// TwinCAT 3 PLC project STELLA1Runtime
// ProgramVersion: 3.1.4023.0
// libraries:
//   Tc2_DataExchange, * (Beckhoff Automation GmbH)
//   Tc2_Math, * (Beckhoff Automation GmbH)
//   Tc2_MC2, * (Beckhoff Automation GmbH)
//   Tc2_MC2_Drive, * (Beckhoff Automation GmbH)
//   Tc2_NC, * (Beckhoff Automation GmbH)
//   Tc2_Standard, * (Beckhoff Automation GmbH)
//   Tc2_System, * (Beckhoff Automation GmbH)
//   Tc2_Utilities, * (Beckhoff Automation GmbH)
//   Tc3_IotBase, * (Beckhoff Automation GmbH)
//   Tc3_Module, * (Beckhoff Automation GmbH)
//   VisuDialogs, * (System)
//   PS_DcUpsEC,2.0,Phoenix Contact GmbH & Co.KG
//   VisuSymbols,3.5.10.0,System
// project tree:
//   DUTs/ E_Blink.TcDUT, E_Horn.TcDUT, E_TCSCommand.TcDUT (not stored), E_TCSErrors.TcDUT (not stored), E_TelescopeMode.TcDUT
//   / GlobalTextList.TcGTLO, PlcTask.TcTTO, Visualization Manager.TcVMO (not stored)
//   GVLs/ GVL_FilterWheel.TcGVL, GVL_Hydraulics.TcGVL (not stored), GVL_Main.TcGVL, GVL_pendant_control.TcGVL, GVL_Safety.TcGVL, GVL_Telescope.TcGVL
//   POUs/ AzimuthElevationControl.TcPOU, CoverControl.TcPOU, DerotatorControl.TcPOU, ElevationControl.TcPOU, FilterWheelControl.TcPOU, FocusControl.TcPOU, HydraulicsControl.TcPOU, MAIN.TcPOU, NasmythControl.TcPOU, PendantControl.TcPOU, SafetyHandling.TcPOU, TelescopeAuxiliary.TcPOU, TelescopeControl.TcPOU, Transformer.TcPOU
//   POUs/FunctionBlocks/ CO_ABERRATION.TcPOU (not stored), CO_REFRACT.TcPOU, FB_ALTAZ2HADEC.TcPOU (not stored), FB_AstroClock.TcPOU (not stored), FB_Axis2.TcPOU, FB_BLINK.TcPOU, FB_ButtonEnable.TcPOU (not stored), FB_Cover.TcPOU, FB_CO_NUTATE.TcPOU, FB_EQ2HOR.TcPOU, FB_EQ2HOR2.TcPOU, FB_EventLog.TcPOU, FB_HADEC2ALTAZ.TcPOU, FB_HOR2EQ.TcPOU, FB_HOR2EQ2.TcPOU (not stored), FB_Horn.TcPOU, FB_InfluxMessage.TcPOU (not stored), FB_LightTimer.TcPOU (not stored), FB_MQTTCommunication.TcPOU, FB_NUTATE.TcPOU (not stored), FB_PRECESS.TcPOU, FB_PRECESS2.TcPOU, FB_PRECESS3.TcPOU, FB_RFTRIG.TcPOU (not stored), FB_SUNPOS.TcPOU (not stored), FB_TimeAverage.TcPOU (not stored), FB_Timer.TcPOU (not stored), FB_TONTP.TcPOU, TelescopeAxisClass.TcPOU
//   POUs/Functions/ ATAN2.TcPOU, CO_REFRACT_FORWARD.TcPOU (not stored), CT2LST.TcPOU (not stored), DateTime2JD.TcPOU, F_Azimuthvelocity.TcPOU, F_DerotatorPosition2.TcPOU, F_Derotatorvelocity.TcPOU, F_Elevationvelocity.TcPOU, F_YREAL.TcPOU, NCError_TO_STRING.TcPOU, PointingModelAzimuth.TcPOU, PointingModelElevation.TcPOU, POLY.TcPOU (not stored), Refraction.TcPOU, TEN.TcPOU
//   VISUs/ Visualization.TcVIS
// real-time tasks:
//   TASK PlcTask: cycle T#10ms, priority 20, ADS port 350
// motion (NC):
//   TASK NC-Task 1 SAF: cycle T#2ms, priority 4, ADS port 501
//   TASK NC-Task 1 SVB: cycle T#10ms, priority 8, ADS port 511
//   AXIS Fokus (id 1)
//     Dynamic: AccelerationMaximum=100, DecelerationMaximum=100, Acceleration=4.5, Deceleration=4.5, Jerk=13.5
//     Velo: RefSearch=0.2, RefSync=0.2, SlowManual=0.1, FastManual=0.5, Maximum=3
//     TargetPosControl: Range=0.1
//     OtherSettings: AllowMotionCmdToSlave=true, PulseDistancePos=1, PulseDistanceNeg=1
//     encoder EncType=4
//       EncPara: ScaleFactorNumerator=0.001, ScaleFactorDenominator=5, MaxCount=#x0000ffff
//         SoftEndMinControl: Enable=true
//         SoftEndMaxControl: Enable=true, Range=100
//         Inc: RefMode=2, RefSoftSyncMask=#x0000ffff
//     drive DrvType=23
//       Analog: VeloReferenz=10.2713178, VeloScale=10, TorqueSetpointScale=10, ScaleFactorActTorque=10
//       TimeComp: TaskDelayCycles=1
//     controller CtrType=1
//       CtrPara: PriorControlFactor=1
//         PosDiffControl: Range=1
//         PID: PosKp=12, CtrlOutputLimit=1
//         Observer: BandWidth=20
//   AXIS Derotator (id 2)
//     General: UnitName=°
//     Dynamic: AccelerationMaximum=20, DecelerationMaximum=20, Acceleration=3.70696, Deceleration=3.70696, Jerk=1.65107
//     Velo: RefSearch=1, RefSync=0.5, SlowManual=0.5, FastManual=5, Fast=11.7222517903646, Maximum=11.7223
//     PositionAreaControl: Range=10
//     TargetPosControl: Range=1, Time=0.1
//     OtherSettings: AllowMotionCmdToSlave=true
//     encoder EncType=8
//       EncPara: ScaleFactorNumerator=0.2, ScaleFactorDenominator=1048576, MaxCount=#xffffffff
//         SoftEndMinControl: Enable=true, Range=-70
//         SoftEndMaxControl: Enable=true, Range=380
//     drive DrvType=9
//       DrvPara: MaxCount=#xffffffff, DriveControlDWord=#x00030100
//         Analog: VeloReferenz=12.894476969401, TorqueSetpointScale=10, ScaleFactorActTorque=0.1
//         TimeComp: TaskDelayCycles=1
//     controller CtrType=1
//       CtrPara: PriorControlFactor=1
//         PosDiffControl: Range=1, Time=0.1
//         Observer: BandWidth=20
//   AXIS Azimuth (id 3)
//     General: UnitName=°
//     Dynamic: AccelerationMaximum=10, DecelerationMaximum=10, Acceleration=3, Deceleration=3, Jerk=1
//     Velo: RefSearch=2, RefSync=1, SlowManual=1, FastManual=5, Fast=798, Maximum=10
//     TargetPosControl: Range=1, Time=0.1
//     OtherSettings: AllowMotionCmdToSlave=true
//     encoder EncType=8
//       EncPara: ScaleFactorNumerator=360, ScaleFactorDenominator=1048576, MaxCount=#xffffffff
//         SoftEndMinControl: Enable=true, Range=-50
//         SoftEndMaxControl: Enable=true, Range=450
//         Inc: RefPosition=180, RefMode=2
//     drive DrvType=9
//       DrvPara: MaxCount=#xffffffff, DriveControlDWord=#x00030100
//         Analog: VeloReferenz=877.8, VeloScale=1.02400649589962, TorqueSetpointScale=10, ScaleFactorActTorque=0.1
//         TimeComp: TaskDelayCycles=1
//     controller CtrType=1
//       CtrPara: PriorControlFactor=1
//         PosDiffControl: Range=3, Time=0.1
//         Observer: BandWidth=20
//   AXIS Elevation (id 4)
//     General: UnitName=°
//     Dynamic: AccelerationMaximum=10, DecelerationMaximum=10, Acceleration=3, Deceleration=3, Jerk=2
//     Velo: RefSearch=0.5, RefSync=0.5, SlowManual=1, FastManual=3, Fast=1026, Maximum=10
//     TargetPosControl: Range=1, Time=0.1
//     OtherSettings: AllowMotionCmdToSlave=true
//     encoder EncType=8
//       EncPara: ScaleFactorNumerator=360, ScaleFactorDenominator=1048576, MaxCount=#xffffffff
//         SoftEndMinControl: Enable=true
//         SoftEndMaxControl: Enable=true, Range=91
//         Inc: RefPosition=73.9885, RefMode=2
//     drive DrvType=9
//       DrvPara: MaxCount=#xffffffff, DriveControlDWord=#x00030100
//         Analog: VeloReferenz=1128.6, VeloScale=1.02400649589962, TorqueSetpointScale=10, ScaleFactorActTorque=0.1
//         TimeComp: TaskDelayCycles=1
//     controller CtrType=1
//       CtrPara: PriorControlFactor=1
//         PosDiffControl: Range=1, Time=0.1
//         Observer: BandWidth=20
//   AXIS FilterWheel (id 5)
//     General: UnitName=°, UnitFlags=#x00000004
//     Dynamic: AccelerationMaximum=1500, DecelerationMaximum=1500, Acceleration=15.2, Deceleration=15.2, Jerk=4.44308
//     Velo: RefSearch=5, RefSync=5, SlowManual=1, FastManual=10, Fast=103.833333333333, Maximum=100
//     TargetPosControl: Range=1
//     OtherSettings: AllowMotionCmdToSlave=true
//     encoder EncType=19
//       EncPara: ScaleFactorNumerator=5, ScaleFactorDenominator=1048576, MaxCount=#xffffffff
//         Inc: RefMode=1, HomingSensorSource=9
//     drive DrvType=16
//       DrvPara: MaxCount=#xffffffff, DriveControlDWord=#x00020000
//         Analog: VeloReferenz=114.216666666667, VeloScale=32, PosScale=5, TorqueSetpointScale=10, ScaleFactorActTorque=0.1
//         TimeComp: TaskDelayCycles=1
//     controller CtrType=1
//       CtrPara: PriorControlFactor=1
//         PosDiffControl: Range=0.2
//         PID: PosKp=3
//         Observer: BandWidth=20
// I/O:
//   DEVICE Gerät 1 (EtherCAT), AmsNetId 5.122.3.233.2.1
//     Klemme 30 (EK1200) [EK1200-5000 EtherCAT Netzteil (2A E-Bus)]
//       Safety Logic (EL6910) [EL6910, TwinSAFE PLC]
//       Safety IN (EL1904) [EL1904, 4 Ch. Safety Input 24V, TwinSAFE]
//         modules: Module 1 (FSOES)
//       Safety OUT (EL2904) [EL2904, 4 Ch. Safety Output 24V, 0.5A, TwinSAFE]
//         modules: Module 1 (FSOES), Module 2 (DO)
//       Power analysis (EL3443) [EL3443 3Ch. Power Measuring]
//       Power0 (EL9410) [EL9410 E-Bus Netzteilklemme (Diagnose)]
//       Main Panel IN (EL1008) [EL1008 8K. Dig. Eingang 24V, 3ms]
//       Hydraulics IN (EL1008) [EL1008 8K. Dig. Eingang 24V, 3ms]
//       Trafo Hydraulics IN (EL1008) [EL1008 8K. Dig. Eingang 24V, 3ms]
//       Main Panel Out (EL2008) [EL2008 8K. Dig. Ausgang 24V, 0.5A]
//       Trafo Hydraulics OUT (EL2008) [EL2008 8K. Dig. Ausgang 24V, 0.5A]
//       Temperature IN (EL3202) [EL3202 2K.Ana. Eingang PT100 (RTD)]
//       Power1 (EL9410) [EL9410 E-Bus Netzteilklemme (Diagnose)]
//       Pendant Control (EL1008) [EL1008 8K. Dig. Eingang 24V, 3ms]
//       Pendant Control2 (EL1008) [EL1008 8K. Dig. Eingang 24V, 3ms]
//       M2 M3 Limit switches (EL1008) [EL1008 8K. Dig. Eingang 24V, 3ms]
//       Cover Limit Switches (EL1008) [EL1008 8K. Dig. Eingang 24V, 3ms]
//       Telescope Hydraulics IN (EL1008) [EL1008 8K. Dig. Eingang 24V, 3ms]
//       Pendant Lights (EL2008) [EL2008 8K. Dig. Ausgang 24V, 0.5A]
//       Lock and Horn (EL2008) [EL2008 8K. Dig. Ausgang 24V, 0.5A]
//       Temperature M2 M1 (EL3064) [EL3064 4K.Ana. Eingang 0-10V]
//       Power2 (EL9410) [EL9410 E-Bus Netzteilklemme (Diagnose)]
//       FocusMotor (EL7342) [EL7342 2K. DC-Motor-Endstufe (50V, 3.5A)]
//       FocusEncoder (EL5101-0010) [EL5101-0010 1K. Inc. Encoder 5V (20 Mio. Inkremente/s)]
//       Cover Motors (EL2008) [EL2008 8K. Dig. Ausgang 24V, 0.5A]
//       Klemme 54 (EK1521) [EK1521 1-Port EtherCAT-Abzweig (FX-MultiMode)]
//         Klemme 55 (EK1501) [EK1501 EtherCAT-Koppler (2A E-Bus, FX-MultiMode, ID-Switch)]
//           FilterWheel (EL7211-0010) [EL7211-0010 1K. MDP742 Servo-Motor-Endstufe mit OCT (50V, 4,5A RMS)]
//           Klemme 57 (EL1008) [EL1008 8K. Dig. Eingang 24V, 3ms]
//           Klemme 58 (EL2008) [EL2008 8K. Dig. Ausgang 24V, 0.5A]
//           ShutterCOM (EL6001) [EL6001 Schnittstelle (RS232)]
//           Klemme 60 (EL3064) [EL3064 4K.Ana. Eingang 0-10V]
//           Klemme 69 (EL3202-0010) [EL3202-0010 2K. Ana. Eingang PT100 (RTD), hochgenau]
//           Klemme 65 (EL9011) [EL9011 Endklemme]
//       Klemme 61 (EK1110) [EK1110 EtherCAT-Verlängerung]
//     Derotator(AX5203-0000-0210) [AX5203-0000-0210 EtherCAT Drive (SoE, 2 Ch.)]
//     Azimuth (AX5125-0000-0214) [AX5125-0000-0214 EtherCAT Drive (SoE, 1 Ch.)]
//     Elevation (AX5125-0000-0214) [AX5125-0000-0214 EtherCAT Drive (SoE, 1 Ch.)]
//     Box 74 (Uninterruptible Power Supply) [QUINT4-UPS/24DC/24DC/40/EC]
// variable links:
//   Device 1 (EtherCAT) <-> Device 1 (EtherCAT)/Term 30 (EK1200)/Safety IN (EL1904)
//     Term 30 (EK1200)/Safety Logic (EL6910)/ConnectionOutputs/TwinSafeGroup1.Safety IN (EL1904) - Module 1 (FSOES)_10 RxPDO <-> Module 1 (FSOES)/TxPDO/FSOE
//   Device 1 (EtherCAT) <-> Device 1 (EtherCAT)/Term 30 (EK1200)/Safety Logic (EL6910)
//     Term 30 (EK1200)/Safety IN (EL1904)/Module 1 (FSOES)/RxPDO/FSOE <-> ConnectionInputs/TwinSafeGroup1.Safety IN (EL1904) - Module 1 (FSOES)_10 TxPDO
//     Term 30 (EK1200)/Safety OUT (EL2904)/Module 1 (FSOES)/TxPDO/FSOE <-> ConnectionOutputs/TwinSafeGroup1.Safety OUT (EL2904) - Module 1 (FSOES)_11 RxPDO
//   Device 1 (EtherCAT) <-> Device 1 (EtherCAT)/Term 30 (EK1200)/Safety OUT (EL2904)
//     Term 30 (EK1200)/Safety Logic (EL6910)/ConnectionInputs/TwinSafeGroup1.Safety OUT (EL2904) - Module 1 (FSOES)_11 TxPDO <-> Module 1 (FSOES)/RxPDO/FSOE
//   NC-Task 1 SAF/Axes/Azimuth <-> Device 1 (EtherCAT)/Azimuth (AX5125-0000-0214)
//     Drive/Inputs/In/nDataIn1 <-> AT/Following distance
//     Drive/Inputs/In/nDcOutputTime <-> InfoData/DcOutputShift
//     Drive/Inputs/In/nState1 <-> AT/Drive status word @bit 8
//     Drive/Inputs/In/nState2 <-> AT/Drive status word
//     Drive/Inputs/In/nState4 @bit 1 <-> WcState/InputToggle
//     Drive/Inputs/In/nState4 <-> WcState/WcState
//     Drive/Outputs/Out/nCtrl1 <-> MDT/Master control word @bit 8
//     Drive/Outputs/Out/nDataOut1 <-> MDT/Position command value
//     Enc/Inputs/In/nDataIn1 <-> AT/Position feedback 1 value
//     Enc/Inputs/In/nDataIn3 <-> AT/Probe value 1 positive edge
//     Enc/Inputs/In/nDcInputTime <-> InfoData/DcInputShift
//     Enc/Inputs/In/nState4 @bit 1 <-> WcState/InputToggle
//     Enc/Inputs/In/nState4 <-> WcState/WcState
//     Enc/Inputs/In/nState5 <-> AT/Probe 1 positive latched
//     Enc/Outputs/Out/nCtrl5 <-> MDT/Probe 1 enable
//   NC-Task 1 SAF/Axes/Derotator <-> Device 1 (EtherCAT)/Derotator(AX5203-0000-0210)
//     Drive/Inputs/In/nDataIn1 <-> AT 1/Following distance
//     Drive/Inputs/In/nDataIn3[0] <-> AT 1/Torque/force feedback value
//     Drive/Inputs/In/nDcOutputTime <-> InfoData/DcOutputShift
//     Drive/Inputs/In/nState1 <-> AT 1/Drive status word @bit 8
//     Drive/Inputs/In/nState2 <-> AT 1/Drive status word
//     Drive/Inputs/In/nState4 @bit 1 <-> WcState/InputToggle
//     Drive/Inputs/In/nState4 <-> WcState/WcState
//     Drive/Outputs/Out/nCtrl1 <-> MDT 1/Master control word @bit 8
//     Drive/Outputs/Out/nDataOut1 <-> MDT 1/Position command value
//     Enc/Inputs/In/nDataIn1 <-> AT 1/Position feedback 1 value
//     Enc/Inputs/In/nDcInputTime <-> InfoData/DcInputShift
//     Enc/Inputs/In/nState4 @bit 1 <-> WcState/InputToggle
//     Enc/Inputs/In/nState4 <-> WcState/WcState
//   NC-Task 1 SAF/Axes/Elevation <-> Device 1 (EtherCAT)/Elevation (AX5125-0000-0214)
//     Drive/Inputs/In/nDataIn1 <-> AT/Following distance
//     Drive/Inputs/In/nDcOutputTime <-> InfoData/DcOutputShift
//     Drive/Inputs/In/nState1 <-> AT/Drive status word @bit 8
//     Drive/Inputs/In/nState2 <-> AT/Drive status word
//     Drive/Inputs/In/nState4 @bit 1 <-> WcState/InputToggle
//     Drive/Inputs/In/nState4 <-> WcState/WcState
//     Drive/Outputs/Out/nCtrl1 <-> MDT/Master control word @bit 8
//     Drive/Outputs/Out/nDataOut1 <-> MDT/Position command value
//     Enc/Inputs/In/nDataIn1 <-> AT/Position feedback 1 value
//     Enc/Inputs/In/nDataIn3 <-> AT/Probe value 1 positive edge
//     Enc/Inputs/In/nDcInputTime <-> InfoData/DcInputShift
//     Enc/Inputs/In/nState4 @bit 1 <-> WcState/InputToggle
//     Enc/Inputs/In/nState4 <-> WcState/WcState
//     Enc/Inputs/In/nState5 <-> AT/Probe 1 positive latched
//     Enc/Outputs/Out/nCtrl5 <-> MDT/Probe 1 enable
//   NC-Task 1 SAF/Axes/FilterWheel <-> Device 1 (EtherCAT)/Term 30 (EK1200)/Term 54 (EK1521)/Term 55 (EK1501)/FilterWheel (EL7211-0010)
//     Drive/Inputs/In/nDcOutputTime <-> InfoData/DcOutputShift
//     Drive/Inputs/In/nState1 <-> DRV Statusword/Statusword
//     Drive/Inputs/In/nState2 <-> DRV Statusword/Statusword @bit 8
//     Drive/Inputs/In/nState4 @bit 1 <-> WcState/InputToggle
//     Drive/Inputs/In/nState4 <-> WcState/WcState
//     Drive/Inputs/In/nState8 <-> DRV Info data 1/Info data 1
//     Drive/Outputs/Out/nCtrl1 <-> DRV Controlword/Controlword
//     Drive/Outputs/Out/nCtrl2 <-> DRV Controlword/Controlword @bit 8
//     Drive/Outputs/Out/nDataOut2 <-> DRV Target velocity/Target velocity
//     Enc/Inputs/In/nDataIn1 <-> FB Position/Position
//     Enc/Inputs/In/nDcInputTime <-> InfoData/DcInputShift
//     Enc/Inputs/In/nState4 @bit 1 <-> WcState/InputToggle
//     Enc/Inputs/In/nState4 <-> WcState/WcState
//   NC-Task 1 SAF/Axes/Fokus <-> Device 1 (EtherCAT)/Term 30 (EK1200)/FocusEncoder (EL5101-0010)
//     Enc/Inputs/In/nDataIn1[0] <-> ENC Status compact/Counter value
//     Enc/Inputs/In/nDataIn2[0] <-> ENC Status compact/Latch value
//     Enc/Inputs/In/nState1 <-> ENC Status compact/Status/Latch C valid
//     Enc/Inputs/In/nState1 @bit 1 <-> ENC Status compact/Status/Latch extern valid
//     Enc/Inputs/In/nState1 @bit 6 <-> ENC Status compact/Status/Open circuit
//     Enc/Inputs/In/nState1 @bit 2 <-> ENC Status compact/Status/Set counter done
//     Enc/Inputs/In/nState1 @bit 5 <-> ENC Status compact/Status/Status of input status
//     Enc/Inputs/In/nState2 @bit 4 <-> ENC Status compact/Status/Status of extern latch
//     Enc/Inputs/In/nState2 <-> ENC Status compact/Status/Status of input A
//     Enc/Inputs/In/nState2 @bit 1 <-> ENC Status compact/Status/Status of input B
//     Enc/Inputs/In/nState2 @bit 2 <-> ENC Status compact/Status/Status of input C
//     Enc/Inputs/In/nState2 @bit 3 <-> ENC Status compact/Status/Status of input gate
//     Enc/Inputs/In/nState2 @bit 5 <-> ENC Status compact/Status/Sync error
//     Enc/Inputs/In/nState2 @bit 6 <-> ENC Status compact/Status/TxPDO State
//     Enc/Inputs/In/nState2 @bit 7 <-> ENC Status compact/Status/TxPDO Toggle
//     Enc/Inputs/In/nState4 @bit 1 <-> WcState/InputToggle
//     Enc/Inputs/In/nState4 <-> WcState/WcState
//     Enc/Outputs/Out/nCtrl1 <-> ENC Control compact/Control/Enable latch C
//     Enc/Outputs/Out/nCtrl1 @bit 3 <-> ENC Control compact/Control/Enable latch extern on negative edge
//     Enc/Outputs/Out/nCtrl1 @bit 1 <-> ENC Control compact/Control/Enable latch extern on positive edge
//     Enc/Outputs/Out/nCtrl1 @bit 2 <-> ENC Control compact/Control/Set counter
//     Enc/Outputs/Out/nDataOut1[0] <-> ENC Control compact/Set counter value
//   NC-Task 1 SAF/Axes/Fokus <-> Device 1 (EtherCAT)/Term 30 (EK1200)/FocusMotor (EL7342)
//     Drive/Inputs/In/nState1 @bit 3 <-> DCM Status Channel 1/Status/Error
//     Drive/Inputs/In/nState1 @bit 5 <-> DCM Status Channel 1/Status/Moving negative
//     Drive/Inputs/In/nState1 @bit 4 <-> DCM Status Channel 1/Status/Moving positive
//     Drive/Inputs/In/nState1 @bit 1 <-> DCM Status Channel 1/Status/Ready
//     Drive/Inputs/In/nState1 <-> DCM Status Channel 1/Status/Ready to enable
//     Drive/Inputs/In/nState1 @bit 6 <-> DCM Status Channel 1/Status/Torque reduced
//     Drive/Inputs/In/nState1 @bit 2 <-> DCM Status Channel 1/Status/Warning
//     Drive/Inputs/In/nState2 @bit 3 <-> DCM Status Channel 1/Status/Digital input 1
//     Drive/Inputs/In/nState2 @bit 4 <-> DCM Status Channel 1/Status/Digital input 2
//     Drive/Inputs/In/nState2 @bit 5 <-> DCM Status Channel 1/Status/Sync error
//     Drive/Inputs/In/nState2 @bit 7 <-> DCM Status Channel 1/Status/TxPDO Toggle
//     Drive/Inputs/In/nState4 @bit 1 <-> WcState/InputToggle
//     Drive/Inputs/In/nState4 <-> WcState/WcState
//     Drive/Outputs/Out/nCtrl1 <-> DCM Control Channel 1/Control/Enable
//     Drive/Outputs/Out/nCtrl1 @bit 2 <-> DCM Control Channel 1/Control/Reduce torque
//     Drive/Outputs/Out/nCtrl1 @bit 1 <-> DCM Control Channel 1/Control/Reset
//     Drive/Outputs/Out/nCtrl1 @bit 3 <-> DCM Control Channel 1/Control/Threshold active
//     Drive/Outputs/Out/nDataOut2[0] <-> DCM Velocity Channel 1/Velocity
//   STELLA1Runtime/STELLA1Runtime Instance <-> Device 1 (EtherCAT)/Azimuth (AX5125-0000-0214)
//     PlcTask Inputs/GVL_Telescope.Azimuth_diagnostic <-> AT/Diagnostic number
//     PlcTask Inputs/GVL_Telescope.Azimuth_inputs <-> AT/Digital inputs, state
//     PlcTask Inputs/GVL_Telescope.Azimuth_torque <-> AT/Torque/force feedback value
//   STELLA1Runtime/STELLA1Runtime Instance <-> Device 1 (EtherCAT)/Box 74 (Uninterruptible Power Supply)
//     PlcTask Inputs/MAIN.arrInputPD @bit {304..432 step 32} <-> TxPDO 1/BATTERY {1..5} ALARMS  (5 links)
//     PlcTask Inputs/MAIN.arrInputPD @bit 80 <-> TxPDO 1/STATUS ACTUAL INPUT CURRENT
//     PlcTask Inputs/MAIN.arrInputPD @bit 64 <-> TxPDO 1/STATUS ACTUAL INPUT VOLTAGE
//     PlcTask Inputs/MAIN.arrInputPD @bit 112 <-> TxPDO 1/STATUS ACTUAL OUTPUT CURRENT 1
//     PlcTask Inputs/MAIN.arrInputPD @bit 96 <-> TxPDO 1/STATUS ACTUAL OUTPUT VOLTAGE 1
//     PlcTask Inputs/MAIN.arrInputPD @bit 128 <-> TxPDO 1/STATUS BATTERY ACTUAL VOLTAGE
//     PlcTask Inputs/MAIN.arrInputPD @bit 144 <-> TxPDO 1/STATUS BATTERY CHARGE CURRENT
//     PlcTask Inputs/MAIN.arrInputPD @bit 160 <-> TxPDO 1/STATUS BATTERY TEMPERATURE
//     PlcTask Inputs/MAIN.arrInputPD @bit 176 <-> TxPDO 1/STATUS DEVICE TEMPERATURE
//     PlcTask Inputs/MAIN.arrInputPD <-> TxPDO 1/STATUS FUNCTIONS
//     PlcTask Inputs/MAIN.arrInputPD @bit 32 <-> TxPDO 1/STATUS INTERFACE
//     PlcTask Inputs/MAIN.arrInputPD @bit 192 <-> TxPDO 1/STATUS SOC REMAINING TIME
//     PlcTask Inputs/MAIN.arrInputPD @bit 224 <-> TxPDO 1/STATUS SOC REMAINING TIME PC SHUTDOWN
//     PlcTask Inputs/MAIN.arrInputPD @bit 240 <-> TxPDO 1/STATUS SOH REMAINING LIFETIME
//     PlcTask Inputs/MAIN.arrInputPD @bit 272 <-> TxPDO 1/UPS DIAGNOSIS ALARMS
//     PlcTask Inputs/MAIN.arrInputPD @bit 256 <-> TxPDO 1/UPS PROCESS ALARMS
//   STELLA1Runtime/STELLA1Runtime Instance <-> Device 1 (EtherCAT)/Derotator(AX5203-0000-0210)
//     PlcTask Inputs/GVL_Telescope.Derotator_diagnostic <-> AT 1/Diagnostic number
//     PlcTask Inputs/GVL_Telescope.Derotator_inputs <-> AT 1/Digital inputs, state
//     PlcTask Inputs/GVL_Telescope.Derotator_torque <-> AT 1/Torque/force feedback value
//   STELLA1Runtime/STELLA1Runtime Instance <-> Device 1 (EtherCAT)/Elevation (AX5125-0000-0214)
//     PlcTask Inputs/GVL_Telescope.Elevation_diagnostic <-> AT/Diagnostic number
//     PlcTask Inputs/GVL_Telescope.Elevation_inputs <-> AT/Digital inputs, state
//     PlcTask Inputs/GVL_Telescope.Elevation_torque <-> AT/Torque/force feedback value
//   STELLA1Runtime/STELLA1Runtime Instance <-> Device 1 (EtherCAT)/Term 30 (EK1200)/Cover Limit Switches (EL1008)
//     PlcTask Inputs/GVL_Telescope.cover1_closed <-> Channel 2/GVL_Telescope.cover1_closed
//     PlcTask Inputs/GVL_Telescope.cover2_closed <-> Channel 4/GVL_Telescope.cover2_closed
//     PlcTask Inputs/GVL_Telescope.cover3_closed <-> Channel 6/GVL_Telescope.cover3_closed
//     PlcTask Inputs/GVL_Telescope.cover1_open <-> Channel 1/GVL_Telescope.cover1_open
//     PlcTask Inputs/GVL_Telescope.cover2_open <-> Channel 3/GVL_Telescope.cover2_open
//     PlcTask Inputs/GVL_Telescope.cover3_open <-> Channel 5/GVL_Telescope.cover3_open
//   STELLA1Runtime/STELLA1Runtime Instance <-> Device 1 (EtherCAT)/Term 30 (EK1200)/Cover Motors (EL2008)
//     PlcTask Outputs/GVL_Telescope.close_cover1 <-> Channel 4/GVL_Telescope.close_cover1
//     PlcTask Outputs/GVL_Telescope.close_cover2 <-> Channel 6/GVL_Telescope.close_cover2
//     PlcTask Outputs/GVL_Telescope.close_cover3 <-> Channel 8/GVL_Telescope.close_cover3
//     PlcTask Outputs/GVL_Telescope.nasmyth_left <-> Channel 1/GVL_Telescope.nasmyth_left
//     PlcTask Outputs/GVL_Telescope.nasmyth_right <-> Channel 2/GVL_Telescope.nasmyth_right
//     PlcTask Outputs/GVL_Telescope.open_cover1 <-> Channel 3/GVL_Telescope.open_cover1
//     PlcTask Outputs/GVL_Telescope.open_cover2 <-> Channel 5/GVL_Telescope.open_cover2
//     PlcTask Outputs/GVL_Telescope.open_cover3 <-> Channel 7/GVL_Telescope.open_cover3
//   STELLA1Runtime/STELLA1Runtime Instance <-> Device 1 (EtherCAT)/Term 30 (EK1200)/Hydraulics IN (EL1008)
//     PlcTask Inputs/GVL_Hydraulics.oil_high <-> Channel 2/GVL_Hydraulics.oil_high
//     PlcTask Inputs/GVL_Hydraulics.oil_low <-> Channel 1/GVL_Hydraulics.oil_low
//     PlcTask Inputs/GVL_Hydraulics.oil_overtemperature <-> Channel 4/GVL_Hydraulics.oil_overtemperature
//     PlcTask Inputs/GVL_Hydraulics.oil_pressure_OK <-> Channel 3/GVL_Hydraulics.oil_pressure_OK
//     PlcTask Inputs/GVL_Hydraulics.oil_undertemperature <-> Channel 5/GVL_Hydraulics.oil_undertemperature
//     PlcTask Inputs/GVL_Hydraulics.oilfilter_dirty <-> Channel 6/GVL_Hydraulics.oilfilter_dirty
//   STELLA1Runtime/STELLA1Runtime Instance <-> Device 1 (EtherCAT)/Term 30 (EK1200)/Lock and Horn (EL2008)
//     PlcTask Outputs/GVL_Telescope.focus_unlock <-> Channel 1/GVL_Telescope.focus_lock
//     PlcTask Outputs/GVL_Telescope.horn <-> Channel 8/GVL_Telescope.horn
//     PlcTask Outputs/GVL_Telescope.nasmyth_lock <-> Channel 2/GVL_Telescope.nasmyth_lock
//   STELLA1Runtime/STELLA1Runtime Instance <-> Device 1 (EtherCAT)/Term 30 (EK1200)/M2 M3 Limit switches (EL1008)
//     PlcTask Inputs/GVL_Telescope.focus_limit_far <-> Channel 2/GVL_Telescope.focus_limit_far
//     PlcTask Inputs/GVL_Telescope.focus_limit_near <-> Channel 1/GVL_Telescope.focus_limit_near
//     PlcTask Inputs/GVL_Telescope.nasmyth_limit_left <-> Channel 3/GVL_Telescope.nasmyth_limit_left
//     PlcTask Inputs/GVL_Telescope.nasmyth_limit_right <-> Channel 4/GVL_Telescope.nasmyth_limit_right
//   STELLA1Runtime/STELLA1Runtime Instance <-> Device 1 (EtherCAT)/Term 30 (EK1200)/Main Panel IN (EL1008)
//     PlcTask Inputs/GVL_Main.key_switch_remote <-> Channel 1/GVL_Main.key_switch_remote
//     PlcTask Inputs/GVL_Main.reset_switch <-> Channel 4/GVL_Main.reset_switch
//     PlcTask Inputs/GVL_Main.start_switch <-> Channel 2/GVL_Main.start_switch
//     PlcTask Inputs/GVL_Main.stop_switch <-> Channel 3/GVL_Main.stop_switch
//   STELLA1Runtime/STELLA1Runtime Instance <-> Device 1 (EtherCAT)/Term 30 (EK1200)/Main Panel Out (EL2008)
//     PlcTask Outputs/GVL_Main.lamp_error <-> Channel 3/GVL_Main.lamp_error
//     PlcTask Outputs/GVL_Main.lamp_on_manual <-> Channel 2/GVL_Main.lamp_ready
//     PlcTask Outputs/GVL_Main.lamp_power <-> Channel 1/GVL_Main.lamp_power
//   STELLA1Runtime/STELLA1Runtime Instance <-> Device 1 (EtherCAT)/Term 30 (EK1200)/Pendant Control (EL1008)
//     PlcTask Inputs/GVL_pendant_control.BCD1 <-> Channel 1/GVL_pendant_control.BCD1
//     PlcTask Inputs/GVL_pendant_control.BCD2 <-> Channel 2/GVL_pendant_control.BCD2
//     PlcTask Inputs/GVL_pendant_control.BCD4 <-> Channel 3/GVL_pendant_control.BCD4
//     PlcTask Inputs/GVL_pendant_control.BCD8 <-> Channel 4/GVL_pendant_control.BCD8
//     PlcTask Inputs/GVL_pendant_control.direction_down <-> Channel 7/GVL_pendant_control.direction_down
//     PlcTask Inputs/GVL_pendant_control.direction_up <-> Channel 6/GVL_pendant_control.direction_up
//     PlcTask Inputs/GVL_pendant_control.key_switch <-> Channel 8/GVL_pendant_control.key_switch
//     PlcTask Inputs/GVL_pendant_control.reset_switch <-> Channel 5/GVL_pendant_control.reset_switch
//   STELLA1Runtime/STELLA1Runtime Instance <-> Device 1 (EtherCAT)/Term 30 (EK1200)/Pendant Control2 (EL1008)
//     PlcTask Inputs/GVL_pendant_control.direction_left <-> Channel 2/GVL_pendant_control.direction_left
//     PlcTask Inputs/GVL_pendant_control.direction_right <-> Channel 3/GVL_pendant_control.direction_right
//     PlcTask Inputs/GVL_pendant_control.start_switch <-> Channel 1/GVL_pendant_control.start_switch
//   STELLA1Runtime/STELLA1Runtime Instance <-> Device 1 (EtherCAT)/Term 30 (EK1200)/Pendant Lights (EL2008)
//     PlcTask Outputs/GVL_pendant_control.lamp_down <-> Channel 2/GVL_pendant_control.lamp_down
//     PlcTask Outputs/GVL_pendant_control.lamp_error <-> Channel 5/GVL_pendant_control.lamp_error
//     PlcTask Outputs/GVL_pendant_control.lamp_left <-> Channel 4/GVL_pendant_control.lamp_left
//     PlcTask Outputs/GVL_pendant_control.lamp_right <-> Channel 3/GVL_pendant_control.lamp_right
//     PlcTask Outputs/GVL_pendant_control.lamp_up <-> Channel 1/GVL_pendant_control.lamp_up
//   STELLA1Runtime/STELLA1Runtime Instance <-> Device 1 (EtherCAT)/Term 30 (EK1200)/Safety Logic (EL6910)
//     PlcTask Inputs/GVL_Safety.Error <-> StandardInputs/TwinSafeGroup1.SafetyError_4
//     PlcTask Inputs/GVL_Safety.State <-> Function Block Info Data/TwinSafeGroup1.Network1.FBEstop1 Info Data/State
//     PlcTask Inputs/GVL_Safety.Stop <-> StandardInputs/TwinSafeGroup1.SafetyStop_7
//     PlcTask Outputs/GVL_Safety.ErrAck <-> StandardOutputs/TwinSafeGroup1.ErrorAcknowledgement_1
//     PlcTask Outputs/GVL_Safety.Restart <-> StandardOutputs/TwinSafeGroup1.RestartSafety_2
//     PlcTask Outputs/GVL_Safety.Run <-> StandardOutputs/TwinSafeGroup1.RunSafety_3
//   STELLA1Runtime/STELLA1Runtime Instance <-> Device 1 (EtherCAT)/Term 30 (EK1200)/Telescope Hydraulics IN (EL1008)
//     PlcTask Inputs/GVL_Hydraulics.oil_reserve <-> Channel 2/GVL_Hydraulics.oil_reserve
//     PlcTask Inputs/GVL_Hydraulics.oilpan_maximum <-> Channel 1/GVL_Hydraulics.oilpan_maximum
//     PlcTask Inputs/GVL_Telescope.azimut_limit_switch <-> Channel 8/GVL_Telescope.azimut_limit_switch
//   STELLA1Runtime/STELLA1Runtime Instance <-> Device 1 (EtherCAT)/Term 30 (EK1200)/Temperature IN (EL3202)
//     PlcTask Inputs/GVL_Main.main_cabinet_temperature <-> RTD Inputs Channel 1/Value
//   STELLA1Runtime/STELLA1Runtime Instance <-> Device 1 (EtherCAT)/Term 30 (EK1200)/Temperature M2 M1 (EL3064)
//     PlcTask Inputs/GVL_Telescope.temperature_mirror1 <-> AI Standard Channel 2/Value
//     PlcTask Inputs/GVL_Telescope.temperature_mirror2 <-> AI Standard Channel 1/Value
//   STELLA1Runtime/STELLA1Runtime Instance <-> Device 1 (EtherCAT)/Term 30 (EK1200)/Term 54 (EK1521)/Term 55 (EK1501)/FilterWheel (EL7211-0010)
//     PlcTask Inputs/GVL_FilterWheel.bCalibrationCam <-> DRV Info data 1/Info data 1
//   STELLA1Runtime/STELLA1Runtime Instance <-> Device 1 (EtherCAT)/Term 30 (EK1200)/Term 54 (EK1521)/Term 55 (EK1501)/Term 60 (EL3064)
//     PlcTask Inputs/TelescopeAuxiliary.raw_dewar_pressure <-> AI Standard Channel 1/Value
//   STELLA1Runtime/STELLA1Runtime Instance <-> Device 1 (EtherCAT)/Term 30 (EK1200)/Trafo Hydraulics IN (EL1008)
//     PlcTask Inputs/GVL_Hydraulics.pump_running <-> Channel 7/GVL_Hydraulics.pump_running
//     PlcTask Inputs/GVL_Hydraulics.suction_running <-> Channel 8/GVL_Hydraulics.suction_running
//     PlcTask Inputs/GVL_Main.brake_clearing <-> Channel 3/GVL_Main.brake_clearing
//     PlcTask Inputs/GVL_Main.trafo_bypassed <-> Channel 2/GVL_Main.trafo_bypassed
//   STELLA1Runtime/STELLA1Runtime Instance <-> Device 1 (EtherCAT)/Term 30 (EK1200)/Trafo Hydraulics OUT (EL2008)
//     PlcTask Outputs/GVL_Hydraulics.oil_pump_enable <-> Channel 1/GVL_Hydraulics.oil_pump_enable
//     PlcTask Outputs/GVL_Hydraulics.oil_suction_enable <-> Channel 2/GVL_Hydraulics.oil_suction_enable
//     PlcTask Outputs/GVL_Main.softstart_trafo <-> Channel 8/GVL_Main.softstart_trafo
//     PlcTask Outputs/GVL_Telescope.brake_azimuth_eve <-> Channel 3/GVL_Telescope.brake_azimuth_eve
//   STELLA1Runtime/STELLA1Runtime Instance <-> NC-Task 1 SAF/Axes/Azimuth
//     PlcTask Inputs/GVL_Telescope.AzimuthAxisRef.NcToPlc <-> Outputs/ToPlc
//     PlcTask Outputs/GVL_Telescope.AzimuthAxisRef.PlcToNc <-> Inputs/FromPlc
//   STELLA1Runtime/STELLA1Runtime Instance <-> NC-Task 1 SAF/Axes/Derotator
//     PlcTask Inputs/GVL_Telescope.DerotatorAxisRef.NcToPlc <-> Outputs/ToPlc
//     PlcTask Outputs/GVL_Telescope.DerotatorAxisRef.PlcToNc <-> Inputs/FromPlc
//   STELLA1Runtime/STELLA1Runtime Instance <-> NC-Task 1 SAF/Axes/Elevation
//     PlcTask Inputs/GVL_Telescope.ElevationAxisRef.NcToPlc <-> Outputs/ToPlc
//     PlcTask Outputs/GVL_Telescope.ElevationAxisRef.PlcToNc <-> Inputs/FromPlc
//   STELLA1Runtime/STELLA1Runtime Instance <-> NC-Task 1 SAF/Axes/FilterWheel
//     PlcTask Inputs/GVL_FilterWheel.FilterWheel_AxisRef.NcToPlc <-> Outputs/ToPlc
//     PlcTask Outputs/GVL_FilterWheel.FilterWheel_AxisRef.PlcToNc <-> Inputs/FromPlc
//   STELLA1Runtime/STELLA1Runtime Instance <-> NC-Task 1 SAF/Axes/Fokus
//     PlcTask Inputs/GVL_Telescope.FocusAxisRef.NcToPlc <-> Outputs/ToPlc
//     PlcTask Outputs/GVL_Telescope.FocusAxisRef.PlcToNc <-> Inputs/FromPlc

CONFIGURATION STELLA1Runtime
    RESOURCE PLC ON TwinCAT3
        TASK PlcTask(INTERVAL := T#10ms, PRIORITY := 20);
        PROGRAM MAIN WITH PlcTask : MAIN;
    END_RESOURCE
END_CONFIGURATION

// ---- DUTs/E_Blink.TcDUT
{attribute 'qualified_only'}
{attribute 'strict'}
TYPE E_Blink :
(
	off := 0,
	slow,
	fast,
	short,
	long,
	on
);
END_TYPE

// ---- DUTs/E_Horn.TcDUT
{attribute 'qualified_only'}
{attribute 'strict'}
TYPE E_Horn :
(
	off := 0,
	beep,
	short,
	long
);
END_TYPE

// ---- DUTs/E_TelescopeMode.TcDUT
{attribute 'qualified_only'}
{attribute 'strict'}
TYPE E_TelescopeMode :
(
	off := 0,
	manual := 1,
	automatic := 2
);
END_TYPE

// ---- GVLs/GVL_FilterWheel.TcGVL
{attribute 'qualified_only'}
VAR_GLOBAL
	FilterWheel_AxisRef:	AXIS_REF;
	bCalibrationCam			AT%I*:	BOOL;
END_VAR

// ---- GVLs/GVL_Main.TcGVL
{attribute 'qualified_only'}
//TODO update to current RoboTel IOs
VAR_GLOBAL
	//DIN1 0.0
	//phase_available		AT%I*: BOOL;
	// not implemented on stella
	trafo_bypassed		AT%I*: BOOL;
	//not implemented on RoboTel
	//key_switch			AT%I*: BOOL;
	//DIN3 0.2
	key_switch_remote	AT%I*: BOOL;
	//DIN4 0.3
	start_switch		AT%I*: BOOL;
	//DIN5 0.4
	stop_switch			AT%I*: BOOL;
	//DIN8 0.7
	reset_switch		AT%I*: BOOL;
	
	//BT1
	main_cabinet_temperature	AT%I*: INT;
	//DIN15 1.6
	brake_clearing		AT%I*: BOOL;
	
	//DOUT1 0.0
	lamp_power			AT%Q*: BOOL;
	//DOUT2 0.1
	lamp_on_manual			AT%Q*: BOOL;
	//DOUT3 0.2
	lamp_error			AT%Q*: BOOL;
	
	//DOUT7 0.6
	softstart_trafo		AT%Q*:BOOL;

	isRoboTel:		BOOL;
END_VAR

// ---- GVLs/GVL_pendant_control.TcGVL
{attribute 'qualified_only'}
//TODO update to current RoboTel IOs
VAR_GLOBAL
	//DIN17 2.0
	BCD1		AT%I*: BOOL;
	//DIN18 2.1
	BCD2		AT%I*: BOOL;
	//DIN19 2.2
	BCD4		AT%I*: BOOL;
	//DIN20 2.3
	BCD8		AT%I*: BOOL;
	//DIN21 2.4
	reset_switch	AT%I*: BOOL;
	//DIN22 2.5
	direction_up	AT%I*: BOOL;
	//DIN23 2.6
	direction_down	AT%I*: BOOL;
	//DIN24 2.7
	key_switch		AT%I*: BOOL;
	//DIN25 3.0 (enable)
	start_switch	AT%I*: BOOL;
	//DIN26 3.1
	direction_left	AT%I*: BOOL;
	//DIN27 3.2
	direction_right	AT%I*: BOOL;
	
	// Outputs
	
	//DOUT9 1.0
	lamp_up			AT%Q*: BOOL;
	//DOUT10 1.1
	lamp_down			AT%Q*: BOOL;
	//DOUT11 1.2
	lamp_right			AT%Q*: BOOL;
	//DOUT12 1.3
	lamp_left			AT%Q*: BOOL;
	//DOUT13 1.4
	lamp_error			AT%Q*: BOOL;
	
END_VAR

// ---- GVLs/GVL_Safety.TcGVL
{attribute 'qualified_only'}
VAR_GLOBAL
	// Safety Error Condition
	Error		AT%I*:	BOOL;
	// Run/Stop Safety
	Run			AT%Q*:	BOOL;
	// Restart Safety
	Restart		AT%Q*:	BOOL;
	// Error Acknowledgement 
	ErrAck		AT%Q*:	BOOL;
	// Stop signal coming from Safety
	Stop		AT%I*:	BOOL;
END_VAR

// ---- GVLs/GVL_Telescope.TcGVL
{attribute 'qualified_only'}
VAR_GLOBAL
	// BT9 mirror
	temperature_mirror2		AT%I*: INT;
	// BT10
	temperature_mirror1		AT%I*: INT;

	//DOUT6 0.5
	brake_azimuth_eve	AT%Q*: BOOL;
	
	// DIN28 3.3 (absolute)
	azimut_limit_switch	AT%I*: BOOL;
	// DIN29 3.4
	focus_limit_near	AT%I*: BOOL;
	// DIN30 3.5
	focus_limit_far		AT%I*: BOOL;
	// DIN31 3.6
	nasmyth_limit_left	AT%I*: BOOL;
	// DIN32 3.7
	nasmyth_limit_right	AT%I*: BOOL;
	
	// DIN33 4.0
	cover1_open		AT%I*: BOOL;
	// DIN34 4.1
	cover1_closed	AT%I*: BOOL;
	// DIN35 4.2
	cover2_open		AT%I*: BOOL;
	// DIN36 4.3
	cover2_closed	AT%I*: BOOL;
	// DIN37 4.4
	cover3_open		AT%I*: BOOL;
	// DIN38 4.5
	cover3_closed	AT%I*: BOOL;

	//DOUT14 1.5
	focus_unlock		AT%Q*: BOOL;
	//DOUT15 4.6
	nasmyth_lock	AT%Q*: BOOL;
	//Horn 4.7
	horn			AT%Q*: BOOL;
	
	// digitale inputs der Endlagen
	Derotator_inputs		AT%I*: WORD;
	// diagnostic number
	Derotator_diagnostic	AT%I*: UDINT;
	// derotator torque feedback
	Derotator_torque		AT%I*: INT;
	
	// digital inputs for limit switches
	Elevation_inputs		AT%I*: WORD;
	// diagnostic number
	Elevation_diagnostic	AT%I*: UDINT;
	// torque feedback
	Elevation_torque		AT%I*: INT;
	
	// digital inputs for limit switches
	Azimuth_inputs			AT%I*: WORD;
	// diagnostic number
	Azimuth_diagnostic		AT%I*: UDINT;
	// torque feedback
	Azimuth_torque			AT%I*: INT;
	
	// Zyklisches Interface zwischen NC und Achse
	AzimuthAxisRef: 	AXIS_REF;
	ElevationAxisRef: 	AXIS_REF;
	DerotatorAxisRef: 	AXIS_REF;
 	// Motor1 Channel 1
	FocusAxisRef:		AXIS_REF;
	
	nasmyth_left	AT%Q*: BOOL;
	nasmyth_right	AT%Q*: BOOL;
	open_cover1		AT%Q*: BOOL;
	close_cover1	AT%Q*: BOOL;
	open_cover2		AT%Q*: BOOL;
	close_cover2	AT%Q*: BOOL;
	open_cover3		AT%Q*: BOOL;
	close_cover3	AT%Q*: BOOL;
	
	
END_VAR

// ---- POUs/MAIN.TcPOU
PROGRAM MAIN
VAR
	// telescope drives are ready to enable
	ready:				BOOL;
	// error stat on drive, power or hydraulics
	error:				BOOL;
	// manual, panel or remote reset
	reset:				BOOL;
	// start hydraulics
	start:				BOOL;
	// stop hydraulics 
	stop:				BOOL;
	// soft start trafo
	key_switch:			BOOL;
	//	open brake
	brake_clearing:		BOOL := FALSE;
	
	remote_start:		BOOL;
	remote_stop: 		BOOL;
	remote_reset:		BOOL;
	remote_keyswitch:	BOOL;
	remote_brake_clearing:	BOOL;
	// blink error lamp on warning
	error_lamp: 		FB_BLINK;
	power_lamp:			FB_BLINK;
	sound_horn:			FB_Horn;
	// main cabinet temperature in degrees
	cabinet_temperature:	REAL;
	// measures time between soft start command and power available
	ups_output_voltage:		REAL;
	ups_output_current:		REAL;
	ups_output_power:		REAL;
	PhaseLog:				FB_EventLog;
	TemperatureEvent,
	TemperatureCriticalEvent:	FB_EventLog;
	MQTTTimer : 		TON := (PT:=T#5S);
	GetHostName:		FB_GetHostName;
	HostName: 			STRING(255);
//	LightSwitch:		FB_ButtonEnable;
//	Lightbutton: 		BOOL;
	bExecute:			BOOL := TRUE;
	cabinet_temperature_warning:	SR;
	cabinet_temperature_critical:	SR;
	MQTTClient:		FB_MQTTCommunication;
	ups: 				PS_Q4_DcUpsEC_Cyclic_2;
	xActivate:			BOOL := TRUE;
	arrInputPD	AT%I*:	ARRAY[0..30] OF WORD;
	UPS_Error,
	UPS_Alarm,
	UPS_Warning,
	UPS_BatMode,
	UPS_ReplaceBattery:	FB_EventLog;
END_VAR

(* 
Main control loop
* Execute sub modules
* power management
* control panel switches and status lamps

* start switch activates Hydraulics and Trafo
* 
*)
GetHostName(bExecute := bExecute, sHostName => HostName);
bExecute := FALSE;
start := GVL_Main.start_switch OR remote_start;
stop := (NOT GVL_Main.stop_switch) OR remote_stop;
key_switch := GVL_Main.key_switch_remote OR remote_keyswitch;
brake_clearing := GVL_Main.brake_clearing OR remote_brake_clearing;
reset := GVL_Main.reset_switch OR GVL_pendant_control.reset_switch OR remote_reset;		
brake_clearing := NOT GVL_Main.brake_clearing;
cabinet_temperature := INT_TO_REAL(GVL_Main.main_cabinet_temperature) / 10.0;
cabinet_temperature_warning(SET1 := cabinet_temperature > 50.0,
							RESET := cabinet_temperature < 40.0);
cabinet_temperature_critical(SET1 := cabinet_temperature > 60.0,
							RESET := cabinet_temperature < 50.0);
IF key_switch THEN
	Transformer.start();
ELSE
	Transformer.stop();
END_IF

IF reset THEN
	Transformer.reset();
END_IF

IF start THEN
	HydraulicsControl.enable := TRUE;
END_IF
IF stop THEN
	HydraulicsControl.enable := FALSE;
END_IF

// telescope is ready when power available
ready :=  GVL_main.trafo_bypassed;

// QUINT UPS control section
ups(
	xActivate:= xActivate, 
	arrInputPD:= arrInputPD, 
	xActive=> , 
	xError=> , 
	wDiagCode=> , 
	wAddDiagCode=> , 
	wOutputVoltage=> ups_output_voltage, 
	wOutputCurrent=> ups_output_current, 
	xBatModeActive=> , 
	udtDataStruct=> , 
	xAlarm=> , 
	xWarning=> , 
	xReplaceBattery=> , 
	udtDiag=> );
	
ups_output_voltage := ups_output_voltage / 1000.0;
ups_output_current := ups_output_current / 1000.0;
ups_output_power := ups_output_voltage * ups_output_current;
		
TelescopeControl();	//
CoverControl();	//
PendantControl();	//
NasmythControl();	//
HydraulicsControl();	//
ElevationControl();	//
AzimuthElevationControl();	//
DerotatorControl();	//
FilterWheelControl();	//
FocusControl();
MQTTClient();
Transformer();

error := GVL_Telescope.azimut_limit_switch
			OR FilterWheelControl.Error
			OR Focuscontrol.Error
			OR NasmythControl.error
			OR CoverControl.Error;
// set control lights					
GVL_Main.lamp_on_manual := PendantControl.manual;

IF GVL_Safety.Error THEN
	error_lamp.blink := e_blink.short;
ELSIF ElevationControl.error OR AzimuthElevationControl.error OR DerotatorControl.Error THEN
	error_lamp.blink := e_blink.long;
ELSIF HydraulicsControl.oil_warning OR HydraulicsControl.oil_hot OR HydraulicsControl.pressure_failure THEN
	error_lamp.blink := e_blink.slow;
ELSIF Transformer.error THEN
	error_lamp.blink := e_blink.fast;
ELSIF error THEN
	error_lamp.blink := e_blink.on;
ELSE
	error_lamp.blink := e_blink.off; 
END_IF

IF Transformer.restart_inhibited THEN
	power_lamp.blink := e_blink.short;
ELSIF GVL_main.trafo_bypassed THEN 
	power_lamp.blink := e_blink.on;
ELSIF Transformer.phase_available THEN
	power_lamp.blink := e_blink.long;
ELSIF NOT Transformer.phase_available THEN
	power_lamp.blink := e_blink.off;
ELSIF  Transformer.error THEN
	power_lamp.blink := e_blink.fast;
ELSE 
	power_lamp.blink := e_blink.off; 
END_IF
error_lamp(Q => GVL_Main.lamp_error);
//GVL_Main.lamp_error := error_lamp.Q;
power_lamp(Q => GVL_Main.lamp_power);
//GVL_Main.lamp_power := power_lamp.Q;

IF GVL_Telescope.azimut_limit_switch THEN
	sound_horn.horn := E_horn.long;
ELSIF Hydraulicscontrol.suction_failure THEN
	sound_horn.horn := E_horn.long;
ELSIF TelescopeControl.poweronwarning.Q THEN
	sound_horn.horn := E_horn.short;
ELSIF Pendantcontrol.horn THEN
	sound_horn.horn := E_horn.beep;
ELSE
	sound_horn.horn := E_horn.off;
END_IF 

sound_horn(Q => GVL_Telescope.horn );

SafetyHandling();

MQTTTimer(IN:=TRUE);
IF MQTTTimer.Q THEN // publish new payload every second
	MQTTTimer(IN:=FALSE);
	MQTTClient.Publish('electronics', 'base', 'MainCabinetTemperature', LREAL_TO_FMTSTR(cabinet_temperature, 2, TRUE));
	MQTTClient.Publish('electronics', 'base', 'PowerOK', BOOL_TO_STRING(Transformer.power_ok));
	MQTTClient.Publish('electronics', 'base', 'PhaseOK', BOOL_TO_STRING(Transformer.phase_available));
	MQTTClient.Publish('electronics', 'base', 'MainReady', BOOL_TO_STRING(ready));
	MQTTClient.Publish('electronics', 'base', 'MasterError', BOOL_TO_STRING(error));
	MQTTClient.Publish('electronics', 'base', 'UPSOutputVoltage', LREAL_TO_FMTSTR(ups_output_voltage, 3, TRUE));
	MQTTClient.Publish('electronics', 'base', 'UPSOutputCurrent', LREAL_TO_FMTSTR(ups_output_current, 3, TRUE));
	MQTTClient.Publish('electronics', 'base', 'UPSOutputPower', LREAL_TO_FMTSTR(ups_output_power, 3, TRUE));
	MQTTClient.Publish('electronics', 'base', 'UpsError', BOOL_TO_STRING(ups.xError));
	MQTTClient.Publish('electronics', 'base', 'UpsAlarm', BOOL_TO_STRING(ups.xAlarm));
	MQTTClient.Publish('electronics', 'base', 'UpsWarning', BOOL_TO_STRING(ups.xWarning));
	MQTTClient.Publish('electronics', 'base', 'UpsBatteryMode', BOOL_TO_STRING(ups.xBatModeActive));
	MQTTClient.Publish('electronics', 'base', 'UPSReplaceBattery', BOOL_TO_STRING(ups.xReplaceBattery));
END_IF

PhaseLog(	
	Trigger := 		NOT Transformer.phase_available, 
	Level := 		ADSLOG_MSGTYPE_ERROR,
	FormatString :=	'%s',
	OnMessage := 	'electrical phases:	ERROR!',
	OffLevel := 	ADSLOG_MSGTYPE_HINT,
	OffMEssage := 	'electrical phases:	active');
	
TemperatureEvent(	
	Trigger := 		cabinet_temperature_warning.Q1, 
	Level := 		ADSLOG_MSGTYPE_WARN,
	FormatString :=	'Main cabinet temperature warning:	%s',
	OnMessage := 	LREAL_TO_FMTSTR( cabinet_temperature, 1, TRUE),);
TemperatureCriticalEvent(	
	Trigger := 		cabinet_temperature_critical.Q1, 
	Level := 		ADSLOG_MSGTYPE_ERROR,
	FormatString :=	'Main cabinet temperature is critical:	%s!',
	OnMessage := 	LREAL_TO_FMTSTR( cabinet_temperature, 1, TRUE),);
	
UPS_Error(	
	Trigger := 		ups.xError, 
	Level := 		ADSLOG_MSGTYPE_ERROR,
	OnMessage := 	'UPS has an error!');

UPS_Alarm(	
	Trigger := 		ups.xAlarm, 
	Level := 		ADSLOG_MSGTYPE_ERROR,
	OnMessage := 	'UPS has an alarm!');

	
UPS_Warning(	
	Trigger := 		ups.xWarning, 
	Level := 		ADSLOG_MSGTYPE_WARN,
	OnMessage := 	'UPS has a warning!');

UPS_BatMode(	
	Trigger := 		ups.xBatModeActive, 
	Level := 		ADSLOG_MSGTYPE_WARN,
	OnMessage := 	'UPS is on battery!');

UPS_ReplaceBattery(	
	Trigger := 		ups.xReplaceBattery, 
	Level := 		ADSLOG_MSGTYPE_WARN,
	OnMessage := 	'Replace UPS battery!');

END_PROGRAM

// ---- POUs/FunctionBlocks/FB_BLINK.TcPOU
FUNCTION_BLOCK FB_BLINK
VAR_INPUT
	blink:		E_Blink;
	ON_TIME:	TIME := T#500MS;
	OFF_TIME:	TIME := T#500MS;
END_VAR
VAR_OUTPUT
	Q:		BOOL;
END_VAR
VAR
    IMPULS   :TOF;
    PAUSE    :TOF;
END_VAR

CASE blink OF
	e_blink.off:
		ON_TIME := T#0MS;
		OFF_TIME := T#1000MS;
	e_blink.slow:
		ON_TIME := T#500MS;
		OFF_TIME := T#500MS;
	e_blink.fast:
		ON_TIME := T#250MS;
		OFF_TIME := T#250MS;
	e_blink.short:
		ON_TIME := T#100MS;
		OFF_TIME := T#900MS;
	e_blink.long:
		ON_TIME := T#900MS;
		OFF_TIME := T#100MS;
	e_blink.on:
		ON_TIME := T#0MS;
		OFF_TIME := T#0MS;
END_CASE

IMPULS(IN:= NOT PAUSE.Q AND NOT IMPULS.Q, PT:= ON_TIME);
PAUSE(IN:= NOT PAUSE.Q AND NOT IMPULS.Q, PT:= OFF_TIME);
IF blink = e_blink.off THEN
	Q := FALSE;
ELSIF blink = e_blink.on THEN
	Q := TRUE;
ELSE
	Q := IMPULS.Q;	
END_IF

END_FUNCTION_BLOCK

// ---- POUs/FunctionBlocks/FB_Horn.TcPOU
FUNCTION_BLOCK FB_Horn
VAR_INPUT
	horn:	E_Horn;
END_VAR
VAR_OUTPUT
		Q:		BOOL;
END_VAR
VAR
	ON_TIME:	TIME := T#500MS;
	IMPULS   :TOF;
    PAUSE    :TOF;

END_VAR

CASE horn OF
	e_horn.off:
		ON_TIME := T#0MS;
	e_horn.beep:
		ON_TIME := T#500MS;
	e_horn.short:
		ON_TIME := T#3000MS;
	e_horn.long:
		ON_TIME := T#5000MS;
END_CASE

IMPULS(IN:= NOT PAUSE.Q AND NOT IMPULS.Q, PT:= ON_TIME);
IF horn = e_horn.off THEN
	Q := FALSE;
ELSE
	Q := IMPULS.Q;	
END_IF

END_FUNCTION_BLOCK

// ---- POUs/FunctionBlocks/FB_EventLog.TcPOU
FUNCTION_BLOCK FB_EventLog
VAR_INPUT
	Trigger:		BOOL;
	// ADSLOG_MSGTYPE_HINT or ADSLOG_MSGTYPE_WARN or ADSLOG_MSGTYPE_ERROR
	Level:			UDINT := ADSLOG_MSGTYPE_HINT;
	FormatString: 	STRING(255) := '%s';
	OnMessage: 		STRING(255) := '';
	OffMessage:		STRING(255) := '';
	OffLevel:		UDINT := ADSLOG_MSGTYPE_HINT;
END_VAR
VAR_OUTPUT
END_VAR
VAR
	LogonTrigger: R_TRIG;
	LogoffTrigger: F_TRIG; // R_Trig or F_Trig ?!
	sPayloadPub, PayloadMessage: STRING(255);
	fbFormat:	FB_FormatString;
END_VAR

LogonTrigger(CLK := Trigger);
LogoffTrigger(CLK := Trigger);
// in case the OffLevel is not set use the default Level Value
IF OffLevel = 0 THEN
	OffLevel := Level;
END_IF
IF LogonTrigger.Q AND LEN(OnMessage)>0 THEN
	ADSLOGSTR( Level OR ADSLOG_MSGTYPE_LOG, FormatString, OnMessage);
END_IF

IF LogoffTrigger.Q AND LEN(OffMessage)>0 THEN
	ADSLOGSTR( OffLevel OR ADSLOG_MSGTYPE_LOG, FormatString, OffMessage);
END_IF

sPayloadPub := 'log,host=CX-22747A';

IF LogonTrigger.Q AND LEN(OnMessage)>1 THEN
	IF Level=ADSLOG_MSGTYPE_HINT THEN
		sPayloadPub := CONCAT(sPayloadPub, ',level=INFO');
	ELSIF Level=ADSLOG_MSGTYPE_WARN THEN
		sPayloadPub := CONCAT(sPayloadPub, ',level=WARNING');
	ELSE
	    sPayloadPub := CONCAT(sPayloadPub, ',level=ERROR');
	END_IF
	fbFormat( sFormat := FormatString, arg1 := F_STRING(OnMessage), sOut => PayloadMessage);
	sPayloadPub := APPEND(sPayloadPub, ' message="', PayloadMessage);
	sPayloadPub := CONCAT(sPayloadPub, '"');
	MQTTCommunication.fbMqttClient.Publish(	
					sTopic:= 'STELLA1/Log', 
					pPayload:= ADR(sPayloadPub), 
					nPayloadSize:= LEN2(ADR(sPayloadPub)),
					eQoS:= TcIotMqttQos.AtMostOnceDelivery,
					bRetain:= FALSE, 
					bQueue:= FALSE );
END_IF

IF LogoffTrigger.Q AND LEN(OffMessage)>1 THEN
	IF OffLevel=ADSLOG_MSGTYPE_HINT THEN
		sPayloadPub := CONCAT(sPayloadPub, ',level=INFO');
	ELSIF OffLevel=ADSLOG_MSGTYPE_WARN THEN
		sPayloadPub := CONCAT(sPayloadPub, ',level=WARNING');
	ELSE
	    sPayloadPub := CONCAT(sPayloadPub, ',level=ERROR');
	END_IF
	
	fbFormat( sFormat := FormatString, arg1 := F_STRING(OffMessage), sOut => PayloadMessage);
	sPayloadPub := APPEND(sPayloadPub, ' message="', PayloadMessage);
	sPayloadPub := CONCAT(sPayloadPub, '"');
	MQTTCommunication.fbMqttClient.Publish(	
					sTopic:= 'STELLA1/Log', 
					pPayload:= ADR(sPayloadPub), 
					nPayloadSize:= LEN2(ADR(sPayloadPub)),
					eQoS:= TcIotMqttQos.AtMostOnceDelivery,
					bRetain:= FALSE, 
					bQueue:= FALSE );
END_IF

END_FUNCTION_BLOCK

// ---- POUs/FunctionBlocks/FB_MQTTCommunication.TcPOU
FUNCTION_BLOCK FB_MQTTCommunication
VAR_INPUT
END_VAR
VAR_OUTPUT
END_VAR
VAR
	GetHostName:		FB_GetHostName;
	HostName: 			STRING(255);
    bSetParameter:		BOOL := FALSE;
    bConnect:			BOOL := FALSE;
    (* received message *)
	bSubscribed: 		BOOL;
	sTopicSub: 			STRING(255) := 'STELLA1/Telescope/SET';
	{attribute 'TcEncoding':='UTF-8'}
	sTopicRcv: 			STRING(255);
	{attribute 'TcEncoding':='UTF-8'}
	fbMessageQueue:		FB_IotMqttMessageQueue;
    fbMessage:			FB_IotMqttMessage;
	fbMqttClient:		FB_IotMqttClient;
	sPayloadRcv: 		STRING;
	influxMessage:		FB_InfluxMessage;
	measurement, 
	parameter, 
	value:		STRING(255);
END_VAR

(*
MQTT Communication section

Source:
https://infosys.beckhoff.com/english.php?content=../content/1033/tf6701_tc3_iot_communication_mqtt/3518541195.html&id=

*)
IF HostName='' THEN
	GetHostName.bExecute := TRUE;
ELSE
	GetHostName.bExecute := FALSE;
	bSetParameter := TRUE;
END_IF

GetHostName(sHostName => HostName);

// set the parameters once
IF bSetParameter THEN
    bSetParameter               := FALSE;
    fbMqttClient.sHostName      := 'sky.stella.iac.es';
    fbMqttClient.nHostPort      := 1883;
    fbMqttClient.sClientId      := HostName; 
    fbMqttClient.sTopicPrefix   := ''; 
	fbMqttClient.nKeepAlive     := 60; 
    fbMqttClient.ipMessageQueue := fbMessageQueue;
	bConnect := TRUE;
END_IF

// connect to the client
IF NOT fbMqttClient.bConnected THEN
;
END_IF

fbMqttClient.Execute(bConnect);
	
IF fbMqttClient.bConnected THEN
    IF NOT bSubscribed THEN
        bSubscribed := fbMqttClient.Subscribe(sTopic:=sTopicSub, 
												eQoS:=TcIotMqttQos.AtMostOnceDelivery);
    END_IF
END_IF

// receive queued messages
IF fbMessageQueue.nQueuedMessages > 0 THEN
    IF fbMessageQueue.Dequeue(fbMessage:=fbMessage) THEN
        fbMessage.GetTopic(pTopic:=ADR(sTopicRcv), nTopicSize:=SIZEOF(sTopicRcv) );
        fbMessage.GetPayload(pPayload:=ADR(sPayloadRcv), nPayloadSize:=SIZEOF(sPayloadRcv), bSetNullTermination:=TRUE);
		ADSLOGSTR( ADSLOG_MSGTYPE_HINT OR ADSLOG_MSGTYPE_LOG, 'MQTT %s', sPayloadRcv);
		IF sTopicRcv = sTopicSub THEN
			influxMessage(  sPayload := sPayloadRcv, measurement => measurement, parameter => parameter, value => value);
			IF NOT PendantControl.manual AND measurement = 'command' THEN
				IF parameter = 'power' THEN
					TelescopeControl.power := STRING_TO_BOOL(value);
				ELSIF parameter = 'park' THEN
					TelescopeControl.park := STRING_TO_BOOL(value);
				ELSIF parameter = 'gohome' THEN
					TelescopeControl.gohome := STRING_TO_BOOL(value);
				ELSIF parameter = 'track' THEN
					TelescopeControl.track := STRING_TO_BOOL(value);
				ELSIF parameter = 'goto' THEN
					TelescopeControl.goto := STRING_TO_BOOL(value);
				ELSIF parameter = 'slew' THEN
					TelescopeControl.slew := STRING_TO_BOOL(value);
				ELSIF parameter = 'stop' THEN
					TelescopeControl.stop := STRING_TO_BOOL(value);
				ELSIF parameter = 'reset' THEN
					TelescopeControl.reset := STRING_TO_BOOL(value);
				ELSIF parameter = 'masterreset' THEN
					ElevationControl.bSoEReset := STRING_TO_BOOL(value);
					AzimuthElevationControl.bSoEReset := STRING_TO_BOOL(value);
					DerotatorControl.bSoEReset := STRING_TO_BOOL(value);
				ELSIF parameter = 'nasmyth' THEN
					NasmythControl.left := STRING_TO_USINT(value) = 1;
					NasmythControl.right := STRING_TO_USINT(value) = 2;
				ELSIF parameter = 'rightascension' THEN
					TelescopeControl.track := FALSE;
					TelescopeControl.rightascension := STRING_TO_LREAL(value);
				ELSIF parameter = 'declination' THEN
					TelescopeControl.track := FALSE;
					TelescopeControl.declination := STRING_TO_LREAL(value);
				ELSIF parameter = 'elevation' THEN
					TelescopeControl.elevation := STRING_TO_LREAL(value);
				ELSIF parameter = 'azimuth' THEN
					TelescopeControl.azimuth := STRING_TO_LREAL(value);
				ELSIF parameter = 'focus' THEN
					FocusControl.position := STRING_TO_LREAL(value);
				ELSIF parameter = 'filter' THEN
					FilterWheelControl.filter_position := STRING_TO_USINT(value);
				ELSIF parameter = 'derotator' THEN
					TelescopeControl.track := FALSE;
					TelescopeControl.derotator_offset := STRING_TO_LREAL(value);
				ELSIF parameter = 'elevationoffset' THEN
					TelescopeControl.elevation_offset := STRING_TO_LREAL(value);
				ELSIF parameter = 'azimuthoffset' THEN
					TelescopeControl.azimuth_offset := STRING_TO_LREAL(value);
				ELSIF parameter = 'derotatoroffset' THEN
					TelescopeControl.derotator_offset := STRING_TO_LREAL(value);ELSE
					ADSLOGSTR( ADSLOG_MSGTYPE_WARN OR ADSLOG_MSGTYPE_LOG, 'MQTT not understood %s', sPayloadRcv);
				END_IF
			END_IF // measurement
		END_IF // Topic
		sPayloadRcv := '';
    END_IF // Dequeue
END_IF

PROPERTY Error : BOOL
GET
Error := fbMqttClient.bError;
END_GET
END_PROPERTY

METHOD Publish : BOOL
VAR_INPUT
	domain: 	STRING(255) := 'environment';
	location: 	STRING(255) := 'roof';
	parameter:	STRING(255);
	value:		STRING(255);
END_VAR
VAR
	sPayloadPub: STRING(255) := '';
	fbFormat:	FB_FormatString;
	bError:		BOOL;
	nErrID: UDINT;
	retain_message:		BOOL := FALSE;
END_VAR
//sPayloadPub := 'environment,location=roof,host=CX-4E6032 ';
fbFormat( sFormat := '%s,location=%s,host=%s %s=%s', 
			arg1 := F_STRING(domain), 
			arg2 := F_STRING(location), 
			arg3 := F_STRING(HostName),
			arg4 := F_STRING(parameter),
			arg5 := F_STRING(value),
 
			sOut => sPayloadPub,
			bError => bError, 
			nErrID => nErrID );
// retain message if value is boolean
retain_message := value = 'TRUE' OR value = 'FALSE';

Publish := fbMqttClient.Publish(	
				sTopic:= 'STELLA1/Telemetry', 
				pPayload:= ADR(sPayloadPub), 
				nPayloadSize:= LEN2(ADR(sPayloadPub)),
				eQoS:= TcIotMqttQos.AtMostOnceDelivery,
				bRetain:= retain_message, 
				bQueue:= FALSE );
END_METHOD

METHOD PublishLog : BOOL
VAR_INPUT
	level: 	STRING(255) := 'INFO';
	message:	STRING(255);
	
END_VAR
VAR
	sPayloadPub: STRING(255) := '';
	fbFormat:	FB_FormatString;
	bError:		BOOL;
	nErrID: UDINT;
END_VAR
VAR_OUTPUT
	published: BOOL;
END_VAR
//sPayloadPub := 'environment,location=roof,host=CX-4E6032 ';
fbFormat( sFormat := 'log,host=%s,level=%s message="%s"', 
			arg1 := F_STRING(HostName), 
			arg2 := F_STRING(level), 
			arg3 := F_STRING(message),
 
			sOut => sPayloadPub,
			bError => bError, 
			nErrID => nErrID );

published := fbMqttClient.Publish(	
				sTopic:= 'STELLA1/Log', 
				pPayload:= ADR(sPayloadPub), 
				nPayloadSize:= LEN2(ADR(sPayloadPub)),
				eQoS:= TcIotMqttQos.AtMostOnceDelivery,
				bRetain:= FALSE, 
				bQueue:= FALSE );
END_METHOD

END_FUNCTION_BLOCK

// ---- POUs/PendantControl.TcPOU
PROGRAM PendantControl
VAR
	// program selection of the pendant control
	Selection:	UINT;
	// error on the pendant control
	Error:		BOOL;
	// manual switch
	manual:		BOOL;
	//enable button
	enable:		BOOL;
	//reset button
	reset:		BOOL;
	// up button
	up:			BOOL;
	// down button
	down:		BOOL;
	// left button
	left:		BOOL;
	// right button
	right:		BOOL;
	lamp_left:		BOOL;
	lamp_right:		BOOL;
	lamp_up:		BOOL;
	lamp_down:		BOOL;
	lamp_error:		BOOL;
	horn:			BOOL;
	// counter for filter position
	Filter_position:	USINT;
	FocusEnable: 		FB_ButtonEnable;
	DerotatorEnable:	FB_ButtonEnable;
	ElevationEnable: 	FB_ButtonEnable;
	AzimuthEnable: 		FB_ButtonEnable;
	FilterWheelEnable:	FB_ButtonEnable;
	TelescopeControlEnable: 	FB_ButtonEnable;
	HydraulicsEnable: 	FB_ButtonEnable;
	TrackingEnable:			FB_ButtonEnable;
	ResetDelay:	TON;
	TwinCATRestart: TC_Restart;
	up_trigger:	R_TRIG;
	down_trigger:	R_TRIG;	
	// manual or automatic operation of the telescope
	telescope_mode : E_TelescopeMode;	
END_VAR

(* 
This program is responsible for the manual control of the telescope.
all movable parts can be controlled from here. This is mainly for testing and
maintenance.
WARNING! Some of the safety routines are disabled, when operating the telescope manually.
*)
// calculate the value of the selector
Selection := 1*BOOL_TO_UINT(GVL_pendant_control.BCD1) + 
			 2*BOOL_TO_UINT(GVL_pendant_control.BCD2) + 
			 4*BOOL_TO_UINT(GVL_pendant_control.BCD4) +
			 8*BOOL_TO_UINT(GVL_pendant_control.BCD8);

// detect disconnection of the manual controls (should also trigger emergency stop).			 
Error := (Selection = 0);

// disable all the lamps
lamp_left := FALSE;
lamp_right := FALSE;
lamp_up := FALSE;
lamp_down := FALSE;
horn := FALSE;

// clooect the state of all buttons
manual := GVL_pendant_control.key_switch;
enable := GVL_pendant_control.start_switch;
reset := GVL_pendant_control.reset_switch;
up := GVL_pendant_control.direction_up;
down := GVL_pendant_control.direction_down;
left := GVL_pendant_control.direction_left;
right := GVL_pendant_control.direction_right;

up_trigger(CLK := up);
down_trigger(CLK := down);
//R_Enable(CLK := enable);
// the error lamp is the same as the error lamp of the main panel
lamp_error := GVL_Main.lamp_error;
CoverControl.active_cover := 0;


// determine the operation of the telescope based on the switch set
IF manual THEN
	telescope_mode := E_TelescopeMode.manual;
ELSE
	telescope_mode := E_TelescopeMode.automatic;
END_IF

// enable only the selected item and connect lamps and buttons accordingly
CASE Selection OF
	1:	// reserved for Cover1 control
		lamp_up := GVL_Telescope.cover1_open;
		lamp_down := GVL_Telescope.cover1_closed;
		IF manual THEN
			//CoverEnable(SET := enable, Q := CoverControl.enable);
			//CoverControl.active_cover := 1;
			//CoverControl.reset := reset;
			GVL_Telescope.open_cover1 := up AND GVL_Telescope.cover1_open;
			GVL_Telescope.close_cover1 := down AND GVL_Telescope.cover1_closed;
			lamp_error := CoverControl.Cover1_Error;	
		ELSE
			IF down THEN 
				CoverControl.close := TRUE;
			END_IF
			IF up THEN
				CoverControl.open := TRUE;
			END_IF		
		END_IF

	2: // Cover2 control
		lamp_up := GVL_Telescope.cover2_open;
		lamp_down := GVL_Telescope.cover2_closed;
		IF manual THEN
			//CoverEnable(SET := enable, Q := CoverControl.enable);
			//CoverControl.active_cover := 2;
			GVL_Telescope.open_cover2 := up AND GVL_Telescope.cover2_open;
			GVL_Telescope.close_cover2 := down AND GVL_Telescope.cover2_closed;
			lamp_error := CoverControl.Cover2_Error;
		ELSE
			IF down THEN 
				CoverControl.close := TRUE;
			END_IF
			IF up THEN
				CoverControl.open := TRUE;
			END_IF		
		END_IF
 	
	3:  // Cover3 control
		lamp_up := GVL_Telescope.cover3_open;
		lamp_down := GVL_Telescope.cover3_closed;
		IF manual THEN
			//CoverEnable(SET := enable, Q := CoverControl.enable);
			//CoverControl.active_cover := 3;
			GVL_Telescope.open_cover3 := up AND GVL_Telescope.cover3_open;
			GVL_Telescope.close_cover3 := down AND GVL_Telescope.cover3_closed;
			//CoverControl.reset := reset;
			lamp_error := CoverControl.Cover3_Error;
		ELSE
			IF down THEN 
				CoverControl.close := TRUE;
			END_IF
			IF up THEN
				CoverControl.open := TRUE;
			END_IF		
		END_IF
		
	4:	// Nasmyth / mirror M3 control
		lamp_left := NOT GVL_Telescope.nasmyth_limit_left;
		lamp_right := NOT GVL_Telescope.nasmyth_limit_right;
		IF manual THEN
			GVL_Telescope.nasmyth_lock := enable;
			//NasmythEnable(SET := enable, Q := NasmythControl.enable);
			GVL_Telescope.nasmyth_left := left AND NOT GVL_Telescope.nasmyth_limit_left;
			GVL_Telescope.nasmyth_right := right AND NOT GVL_Telescope.nasmyth_limit_right;
			//NasmythControl.left := left;
			//NasmythControl.right := right;
			NasmythControl.reset := reset;
			lamp_error := Nasmythcontrol.error;
		END_IF
		
	5:	// Focus Control
		lamp_up := FocusControl.Ready AND NOT GVL_Telescope.focus_limit_far;
		lamp_down := FocusControl.Ready AND NOT GVL_Telescope.focus_limit_near;
		IF manual THEN
			FocusEnable(SET := enable, Q := FocusControl.enable);
			FocusControl.outward := up;
			FocusControl.inward := down;
			Focuscontrol.reset := reset;
			lamp_error := FocusControl.error;
		END_IF
							
	6:	// Derotator control
		lamp_left := DerotatorControl.Ready AND NOT GVL_Telescope.Derotator_inputs.1;
		lamp_right :=DerotatorControl.Ready AND NOT GVL_Telescope.Derotator_inputs.0;
		IF manual THEN
			DerotatorEnable(SET := enable, Q := DerotatorControl.enable);
			DerotatorControl.left := left AND NOT GVL_Telescope.Derotator_inputs.1;
			DerotatorControl.right := right AND NOT GVL_Telescope.Derotator_inputs.0;
			DerotatorControl.reset := reset;
			lamp_error := DerotatorControl.Error;
		END_IF
							
	7:	// Elevation Control
		
		ElevationControl.up := up AND GVL_Telescope.Elevation_inputs.0;
		ElevationControl.down := down AND GVL_Telescope.Elevation_inputs.1;
		IF manual THEN
			ElevationEnable(
				SET := enable, 
				Q := ElevationControl.enable);	
		END_IF
		ElevationControl.reset := reset;
		lamp_up := GVL_Telescope.Elevation_inputs.0;
		lamp_down := GVL_Telescope.Elevation_inputs.1;
		lamp_error := ElevationControl.error;
		
	8:	// Azimuth Control
		lamp_left := GVL_Telescope.Azimuth_inputs.0; // NOT GVL_Telescope.azimut_limit_switch;
		lamp_right := GVL_Telescope.Azimuth_inputs.1; // NOT GVL_Telescope.azimut_limit_switch;
		AzimuthElevationControl.left := left AND GVL_Telescope.Azimuth_inputs.0;
		AzimuthElevationControl.right := right AND GVL_Telescope.Azimuth_inputs.1;
		AzimuthElevationControl.reset := reset;
		IF manual THEN
			AzimuthEnable(
				SET := enable, 
				Q := AzimuthElevationControl.enable);
			lamp_error := AzimuthElevationControl.error;
		END_IF
		
	9: 	// Dome control
		
		
		
	10:	// FilterWheel control
		lamp_left := manual AND FilterWheelControl.enable;
		lamp_right := manual AND FilterWheelControl.enable;
		lamp_up :=	NOT  manual AND FilterWheelControl.enable AND FilterWheelControl.Calibrated;
		lamp_down := NOT manual AND FilterWheelControl.enable AND FilterWheelControl.Calibrated;
		FilterWheelControl.reset := reset;
		FilterWheelControl.left := left;
		FilterWheelControl.right := right;
		
		IF manual THEN
			FilterWheelEnable(SET := enable, Q := FilterWheelControl.enable);
			IF up_trigger.Q THEN
				Filter_position := (Filter_position + 1) MOD 24;
				FilterWheelControl.filter_position := Filter_position;
			ELSIF down_trigger.Q THEN
				Filter_position := (Filter_position - 1) MOD 24;
				FilterWheelControl.filter_position := Filter_position;
			END_IF
			lamp_error := FilterWheelControl.Error;
		END_IF
		
	11: lamp_up := ElevationControl.elevation_torque > 0.0;
		lamp_down := ElevationControl.elevation_torque < 0.0;
		
	12:	// manual Telescope Control
		IF manual THEN
			lamp_up := TelescopeControl.power;
			lamp_down := TelescopeControl.power;
			lamp_left := TelescopeControl.power;
			lamp_right := TelescopeControl.power;
	
			TelescopeControl.gohome := down;
			TelescopeControl.park := up;
			TelescopeControl.goto := right;
			TrackingEnable(SET := enable, 
							RESET := reset, 
							Q := TelescopeControl.track);
			TelescopeControl.reset := reset;
			Telescopecontrol.stop := left;	
			lamp_error := Telescopecontrol.error;
		END_IF
		
	13: // Telescope Control
		TelescopeControlEnable(
			SET := enable, 
			Q := TelescopeControl.power);
		TelescopeControl.reset := reset;
		IF manual THEN
			lamp_up := GVL_Telescope.Elevation_inputs.0;
			lamp_down := GVL_Telescope.Elevation_inputs.1;
			lamp_left := GVL_Telescope.Azimuth_inputs.0;
			lamp_right := GVL_Telescope.Azimuth_inputs.1;
			ElevationControl.up := up AND GVL_Telescope.Elevation_inputs.0;
			ElevationControl.down := down AND GVL_Telescope.Elevation_inputs.1;
			AzimuthElevationControl.left := left AND GVL_Telescope.Azimuth_inputs.0;
			AzimuthElevationControl.right := right AND GVL_Telescope.Azimuth_inputs.1;
			TelescopeControl.rightascension := TelescopeControl.rightascension_calc;
			TelescopeControl.declination := TelescopeControl.declination_calc;
		ELSE
			lamp_up := ElevationControl.enable;
			lamp_down := ElevationControl.enable;
			lamp_left := AzimuthElevationControl.enable;
			lamp_right := AzimuthElevationControl.enable;
			IF up THEN 
				Telescopecontrol.elevation_offset := Telescopecontrol.elevation_offset + 10.0/3600.0; 
			ELSIF down THEN 
				Telescopecontrol.elevation_offset := Telescopecontrol.elevation_offset - 10.0/3600.0; 
			END_IF;
			IF left THEN 
				Telescopecontrol.azimuth_offset := Telescopecontrol.azimuth_offset - 10.0/3600.0; 
			ELSIF right THEN 
				Telescopecontrol.azimuth_offset := Telescopecontrol.azimuth_offset + 10.0/3600.0; 
			END_IF;
		END_IF
		ResetDelay(IN := reset, PT := T#3S);
		// wait for suction pump to stop
		TwinCATRestart(NETID := '', RESTART := ResetDelay.Q AND NOT HydraulicsControl.suction_running, TMOUT := T#60S);
	
	14: horn := manual;
		lamp_up := manual;
		lamp_down := manual;
		lamp_left := manual;
		lamp_right := manual;
	
	15:	// Hydraulics control
		lamp_up := HydraulicsControl.oil_pressure_OK AND Hydraulicscontrol.brake_closed;
		lamp_down := HydraulicsControl.oil_pressure_OK AND Hydraulicscontrol.brake_open;
		lamp_left := HydraulicsControl.pump_running;
		lamp_right := HydraulicsControl.suction_running;
		IF manual THEN
			HydraulicsEnable(
				SET := enable, 
				Q := Hydraulicscontrol.enable);
			Hydraulicscontrol.reset := reset;
			
			IF up THEN
				Hydraulicscontrol.open_brake();
			END_IF
			IF down THEN
				Hydraulicscontrol.close_brake();
			END_IF
			Hydraulicscontrol.suction_manual := right;
			Hydraulicscontrol.pump_manual_stop := left;
			lamp_error := HydraulicsControl.error;
		END_IF
END_CASE

// set all the lamps
GVL_pendant_control.lamp_left := lamp_left;
GVL_pendant_control.lamp_right := lamp_right;
GVL_pendant_control.lamp_up := lamp_up;
GVL_pendant_control.lamp_down := lamp_down;
GVL_pendant_control.lamp_error := lamp_error;

END_PROGRAM

// ---- POUs/CoverControl.TcPOU
PROGRAM CoverControl
VAR_INPUT
	// enables all cover drivers
	enable:		BOOL;
	// resets all drives after an error has occured
	reset:		BOOL;
	// open the cover in proper order
	open:		BOOL;
	// close the cover in proper order
	close:		BOOL;
	// actual active cover in manual mode, 0 for automatic = all covers active
	active_cover:	INT;

END_VAR
VAR_OUTPUT
	// is TRUE, if all covers are open
	isopen:			BOOL;
	// is TRUE, if all covers are closed
	isclosed:		BOOL;
	// is TRUE if any cover-driver reports an error
	Error: 	BOOL;
	// warning state of the DC drives
	Warning: BOOL;
	// cover1 is open
	Cover1_opened, 
	// cover1 is closed
	Cover1_closed:	BOOL;
	// cover2 is open
	Cover2_opened, 
	// cover2 is closed
	Cover2_closed:	BOOL;
	// cover3 is open
	Cover3_opened, 
	// cover3 is closed
	Cover3_closed:	BOOL;
	Cover1_error: BOOL;
	Cover2_error: BOOL;
	Cover3_error: BOOL;
	Ready:		BOOL;
END_VAR
VAR
	// delay timer for opening cover2
	open2_delay: 	TON := (PT:=T#1S);;
	// dely timer for closing cover3
	close3_delay : 	TON := (PT:=T#3S);;
	
	//error event for cover1
	Cover1_Event,
	Cover2_Event,
	Cover3_Event:	FB_EventLog;
	// timeout event for cover1
	Cover1_Timeout_Event,
	Cover2_Timeout_Event,
	Cover3_Timeout_Event:	FB_EventLog;
	// log if covers are open
	Covers_opened_event,
	// log if covers are closed
	Covers_closed_event:	FB_EventLog;
	// Event log for a generic drive error
	Covers_Error_event:		FB_EventLog;
	// Event log for a generic drive warning
	Covers_Warning_event:		FB_EventLog;
END_VAR

(*
This is the control for the two (three) telescope covers. 
The correct order for opening is 1->3->2 and for closing 2->3->1.
GVL Open and close signals are inverted
*)

// close has precedence over open
IF close THEN
	open := FALSE;
END_IF

Cover1_opened := NOT GVL_Telescope.cover1_open;
Cover2_opened := NOT GVL_Telescope.cover2_open;
Cover3_opened := NOT GVL_Telescope.cover3_open;
Cover1_closed := NOT GVL_Telescope.cover1_closed;
Cover2_closed := NOT GVL_Telescope.cover2_closed;
Cover3_closed := NOT GVL_Telescope.cover3_closed;
Cover1_error := Cover1_opened AND Cover1_closed;
Cover2_error := Cover2_opened AND Cover2_closed;
Cover3_error := Cover3_opened AND Cover3_closed;

// wait for cover2 until cover3 has left the closed state
open2_delay(IN := open AND NOT cover3_closed);
// wait for cover3 until cover2 has left the open state
close3_delay(IN := close AND NOT cover2_opened);

IF close THEN
	GVL_Telescope.close_cover1 := GVL_Telescope.cover1_closed AND NOT GVL_Telescope.cover3_closed;
	GVL_Telescope.close_cover2 := GVL_Telescope.cover2_closed;
	GVL_Telescope.close_cover3 := GVL_Telescope.cover3_closed AND close3_delay.Q;
ELSIF open THEN
	GVL_Telescope.open_cover1 := GVL_Telescope.cover1_open;
	GVL_Telescope.open_cover2 := GVL_Telescope.cover2_open AND open2_delay.Q;
	GVL_Telescope.open_cover3 := GVL_Telescope.cover3_open;			
END_IF


// we are open, if all covers are open
isopen := cover3_opened AND cover2_opened AND cover1_opened;
// we are closed, if all covers are closed
isclosed := cover2_closed AND cover3_closed AND cover1_closed;
// error indicates an axis error on any axis
Error := (Cover1_error AND NOT GVL_Main.isRoboTel) OR Cover2_error OR Cover3_error;
//Warning := Cover1_control.Warning OR Cover2_control.Warning OR Cover3_control.Warning;

IF isclosed THEN
	close := FALSE;
END_IF

IF isopen THEN
	open := FALSE;
END_IF

Covers_Error_Event.OnMessage := 'Cover drive error';
IF Error THEN
	IF Cover3_error THEN 
		Covers_Error_Event.OnMessage := 'Cover 3 has a drive error.';
	END_IF
	IF Cover2_error THEN 
		Covers_Error_Event.OnMessage := 'Cover 2 has a drive error.';
	END_IF
	IF Cover1_error  AND NOT GVL_Main.isRoboTel THEN 
		Covers_Error_Event.OnMessage := 'Cover 1 has a drive error.';
	END_IF
END_IF

Covers_Error_event(	Trigger := Error, 
					Level := ADSLOG_MSGTYPE_ERROR);

Covers_Warning_event(	Trigger := Warning, 
						Level := ADSLOG_MSGTYPE_WARN);

// raise an error, if both opened and closed signals are activated
// handle RoboTel differently
Cover1_Event(	Trigger := cover1_opened AND cover1_closed AND NOT GVL_Main.isRoboTel,
				Level := ADSLOG_MSGTYPE_ERROR, 
				OnMessage := 'Cover1: limit switch error');

Cover2_Event(Trigger := cover2_opened AND cover2_closed,
				Level := ADSLOG_MSGTYPE_ERROR, 
				OnMessage := 'Cover2: limit switch error');

Cover3_Event(Trigger := cover3_opened AND cover3_closed,
				Level := ADSLOG_MSGTYPE_ERROR, 
				OnMessage := 'Cover3: limit switch error');

//trigger an event, if we encounter a timeout
// handle RoboTel differently

Cover1_Timeout_Event(Trigger := FALSE,
				Level := ADSLOG_MSGTYPE_ERROR, 
				OnMessage := 'Cover1: Timeout');

Cover2_Timeout_Event(Trigger := FALSE,
				Level := ADSLOG_MSGTYPE_ERROR, 
				OnMessage := 'Cover2: Timeout');

Cover3_Timeout_Event(Trigger := FALSE,
				Level := ADSLOG_MSGTYPE_ERROR, 
				OnMessage := 'Cover3: Timeout');
// Log if we are opened
Covers_opened_event(Trigger := isopen,
					Level := ADSLOG_MSGTYPE_WARN,
					OnMessage := 'All covers are open');
//log if we are closed
Covers_closed_event(Trigger := isclosed,
					Level := ADSLOG_MSGTYPE_HINT,
					OnMessage := 'All covers are closed');

END_PROGRAM

// ---- POUs/NasmythControl.TcPOU
PROGRAM NasmythControl
VAR_INPUT
	// unlocks the brake and enables the drive
	enable:	BOOL;
	// resets the drive
	reset: BOOL;
	// turns the Nasmyth mirror to left port (seen from top)
	left:	BOOL;
	// turns the Nasmyth mirror to right port (seen from top)
	right:	BOOL;
END_VAR
VAR_OUTPUT
	// Nasmyth drive error
	error:	BOOL;
	// drive ready
	Ready:	BOOL;
	// Nasmyth points to right mirror
	Nasmyth_right:		BOOL;
	// Nasmyth points to left mirror
	Nasmyth_left:		BOOL;
END_VAR
VAR
	// axis function block
	Nasmyth_control:	FB_Cover;
	// delay for the Nasmyth holding brake
	Nasmyth_delay:		TON;
	// status word for MQTT message
	Nasmyth_status:		WORD;
	// last status word to trigger MQTT message if different
	LastStatus:			WORD;
	// unlock the holding brake
	Nasmyth_unlock:		BOOL;
	// holding brake is unlocked
	Nasmyth_unlocked:	BOOL;
	// event log of error
	NasmythEvent: 		FB_Eventlog;
	NasmythLeftEvent:	FB_Eventlog;
	NasmythRightEvent:	FB_Eventlog;
	Nasmyth_Timeout:	TON := (PT := T#10S);
	
END_VAR

// get the inputs
Nasmyth_left := GVL_Telescope.nasmyth_limit_right;
Nasmyth_right := GVL_Telescope.nasmyth_limit_left;

// disable command, if position has been reached or 
IF Nasmyth_left OR right THEN
	left := FALSE;
END_IF

IF  Nasmyth_right OR left THEN
	right := FALSE;
END_IF

Nasmyth_status.0 := Nasmyth_unlocked;
Nasmyth_status.1 := error;
Nasmyth_status.2 := Nasmyth_left;
Nasmyth_status.3 := Nasmyth_right;
Nasmyth_status.4 := Nasmyth_Timeout.Q;
Nasmyth_status.5 := Ready;

Nasmyth_unlock := enable AND (left OR right);
// report Nasmyth unlocked after n milliseconds										
Nasmyth_delay(
	IN := Nasmyth_unlock,
	PT := T#250MS,
	Q => Nasmyth_unlocked);

// set the outputs
IF NOT PendantControl.manual THEN
	GVL_Telescope.nasmyth_lock := Nasmyth_unlock;
	Nasmyth_control(
		open := left,
		close := right,
		enable := Nasmyth_unlocked,
		reset := reset,
		limit_open := NOT Nasmyth_left,
		limit_close := NOT Nasmyth_right,
		error => error,
		Ready => ready);	
END_IF
	


Nasmyth_Timeout(IN := (left AND NOT Nasmyth_left) OR (right AND NOT Nasmyth_right));

IF Nasmyth_status <> LastStatus THEN
	LastStatus := Nasmyth_status;
	MAIN.MQTTClient.Publish('telescope', 'nasmyth', 'NasmythUnlocked', BOOL_TO_STRING(Nasmyth_unlocked));
	MAIN.MQTTClient.Publish('telescope', 'nasmyth', 'NasmythError', BOOL_TO_STRING(error));
	MAIN.MQTTClient.Publish('telescope', 'nasmyth', 'NasmythReady', BOOL_TO_STRING(Ready));
	MAIN.MQTTClient.Publish('telescope', 'nasmyth', 'NasmythIsLeft', BOOL_TO_STRING(Nasmyth_left));
	MAIN.MQTTClient.Publish('telescope', 'nasmyth', 'NasmythIsRight', BOOL_TO_STRING(Nasmyth_right));
END_IF


NasmythEvent(	Trigger := error, 
				Level := ADSLOG_MSGTYPE_ERROR,
				OnMessage := 'Nasmyth axis error',
				OffMessage := 'OK',
				OffLevel := ADSLOG_MSGTYPE_HINT);

NasmythLeftEvent(	Trigger := Nasmyth_left, 
					Level := ADSLOG_MSGTYPE_HINT,
					OnMessage := 'Nasmyth is on left port');

NasmythRightEvent(	Trigger := Nasmyth_right, 
					Level := ADSLOG_MSGTYPE_HINT,
					OnMessage := 'Nasmyth is on right port');

END_PROGRAM

// ---- POUs/FunctionBlocks/FB_Cover.TcPOU
FUNCTION_BLOCK FB_Cover
VAR_INPUT
	open,
	close,
	enable,
	reset,
	limit_open,
	limit_close: 		BOOL;
END_VAR
VAR_OUTPUT
	error:				BOOL;
	Ready:				BOOL;
	Moving_negative:	BOOL;
	Moving_positive:	BOOL;
	timeout:			BOOL;
END_VAR
VAR
	error_state:	SR;
	//triggers for timeout event for cover
	Cover_timeout:	TON;
	open_timeout: TON := (PT := T#3S);
	close_timeout: TON := (PT := T#3S);
END_VAR


error_state(SET1 := limit_open AND limit_close OR timeout,
			RESET := reset,
			Q1 => error);

IF enable THEN
	Moving_positive := open AND NOT limit_open;
	Moving_negative := close AND NOT limit_close;
END_IF
// A timeout occurs, when we open the cover, and the opened signal does not activate within n seconds.
// The same holds for closing the cover. This should not take longer then 10 seconds
Cover_timeout(IN := NOT (limit_open XOR limit_close) AND (open OR close), PT := T#20S);
open_timeout(IN := open AND limit_open, PT := T#3S);
close_timeout(IN := close AND limit_close, PT := T#3S);
timeout := Cover_timeout.Q OR open_timeout.Q OR close_timeout.Q;

Ready := NOT error;

END_FUNCTION_BLOCK

// ---- POUs/FocusControl.TcPOU
PROGRAM FocusControl
VAR_INPUT
	// enable the axis
	enable: BOOL;
	// Move M2 closer to M1
	inward: 	BOOL;
	// Move M2 away from M1
	outward: 	BOOL;	
	// reset the axis(-error)
	reset: 		BOOL;
	// move the axis to new position
	MoveAxis:	BOOL;
	// calibrate the focus axis
	HomeAxis:	BOOL;
	// focus position in millimeters
	position: 		LREAL;
END_VAR

VAR_OUTPUT
	// true if absolute calibration
	Calibrated:	BOOL;
	// true if error
	Error: 		BOOL;
	// ID of NC axis error
	ErrorID:	UDINT;
	// ready signal = drive ready + standstill
	Ready:	BOOL;
END_VAR

VAR
	FocusDelay:			TON;
	BrakeDelay:			TON;
	FocusAxis:			FB_Axis2;
	actual_position:	LREAL;
	// manual override to unlock the focus
	FocusUnlock:		BOOL;
	FocusUnlocked:		BOOL;
	MQTTTimer : 		TON := (PT:=T#5S);
	//getlastposition:	BOOL := TRUE;
	FocusAxisEvent:		FB_EventLog;
	CalibrationEvent:	FB_EventLog;
	HomingMode: 		MC_HOMINGMODE := 		MC_DefaultHoming;
END_VAR

VAR CONSTANT
	// reference position for homing
	homing_position:		LREAL := 92.8936; // 106.5936 - 13.7000
	tolerance:				LREAL := 0.005;
END_VAR
VAR PERSISTENT
	last_position:		LREAL := -1.0;
END_VAR

(*
Focus Control Unit
spindle gear: 5mm
brake: 86 61103H00 Var. 0005 Index C; 24VDC geglattet 0,25 A P1672/R7
motor: Faulhaber ; Schönaich ; 3557K024CR; 454  431 ; Made in germany ==> 5300 rpm
gear: Faulhaber ; MINIMOTOR SA ; swiss made ; 38/1S  43:1 ; 033896  503
Focus is locked by default
70,8W; 0,100A no load current; 2,0 Terminal resistance; 1,950A max Current 
*)
position := LIMIT(5.0, position, 95.0);

GVL_Telescope.focus_unlock := FocusUnlock OR enable;

// wait until the focus is unlocked for n milliseconds
FocusDelay(IN := GVL_Telescope.focus_unlock, PT := T#500MS, Q => FocusUnlocked);
// wait for brake until we are at rest
BrakeDelay(IN := NOT FocusAxis.Busy AND FocusAxis.StandStill, PT := T#4000MS);

// if we are on automatic mode then position the filterwheel
IF Pendantcontrol.telescope_mode = E_TelescopeMode.automatic AND NOT FocusUnlock THEN
	IF FocusAxis.Calibrated THEN
		IF ABS(position - actual_position) > tolerance THEN
			IF FocusAxis.Ready THEN
				MoveAxis := TRUE;
			ELSE
				Enable := TRUE;
			END_IF
		END_IF
		// disable the drive and lock the brake, if we stand for more than n seconds
		IF BrakeDelay.Q THEN
			Enable := FALSE;
		END_IF
		// store actual position, if we are calibrated and locked
		IF NOT GVL_Telescope.focus_unlock THEN
			last_position := actual_position;
		END_IF
	ELSE // not calibrated
		IF FocusAxis.Ready THEN
			HomeAxis := TRUE;
		END_IF
	END_IF
END_IF

IF HomeAxis THEN
	IF last_position > 0.0 THEN
		HomingMode := MC_ForceCalibration; // MC_Direct
		position := last_position;
	ELSE
		HomingMode := MC_DefaultHoming;
		position := homing_position;
	END_IF
		
END_IF

// deactivate limit switches on homing
MC_SetAcceptBlockedDriveSignal(
	Axis := GVL_Telescope.FocusAxisRef, 
	Enable := HomeAxis);

FocusAxis(	
	Enable := 			FocusUnlocked,
	Reset := 			reset,
	MoveAxis := 		MoveAxis AND FocusUnlocked,
	HomeAxis :=			HomeAxis AND FocusUnlocked,
	HomingMode :=		HomingMode,
	Position := 		position,
	Velocity :=			1.0,
	Enable_Positive := 	NOT GVL_Telescope.focus_limit_far OR HomeAxis,
	Enable_Negative := 	NOT GVL_Telescope.focus_limit_near,
	Jog_Forward :=		outward AND FocusUnlocked,
	Jog_Backwards := 	inward AND FocusUnlocked,
	bCalibrationCam :=  GVL_Telescope.focus_limit_far,
	ActualPosition => 	actual_position,
	Error =>			error,
	ErrorID =>			ErrorID,
	AxisRef :=			GVL_Telescope.FocusAxisRef);	

IF FocusAxis.MoveDone THEN
	MoveAxis := FALSE;
END_IF

IF FocusAxis.HomeDone THEN
	HomeAxis := FALSE;
	Enable := FALSE;
	last_position := position;
END_IF
	
IF FocusAxis.ResetDone THEN
	reset := FALSE;
END_IF

IF FocusAxis.Calibrated OR Error THEN
	HomeAxis := FALSE;
END_IF

IF Error THEN
	last_position := -1.0;
END_IF

Calibrated := FocusAxis.Calibrated;

Ready := FocusAxis.Ready AND FocusAxis.StandStill OR NOT GVL_Telescope.focus_unlock;

MQTTTimer(IN:=TRUE);
IF MQTTTimer.Q THEN // publish new payload every second
	MQTTTimer(IN:=FALSE);
	MAIN.MQTTClient.Publish('telescope', 'dome', 'FocusPosition', LREAL_TO_FMTSTR(actual_position, 5, TRUE));
	MAIN.MQTTClient.Publish('telescope', 'dome', 'FocusCalibrated', BOOL_TO_STRING(Calibrated));	
	MAIN.MQTTClient.Publish('telescope', 'dome', 'FocusReady', BOOL_TO_STRING(Ready));	
END_IF

FocusAxisEvent(	
	Trigger := 		FocusAxis.Error, 
	Level := 		ADSLOG_MSGTYPE_ERROR,
	FormatString :=	'Focus Axis Error: %s',
	OnMessage := 	NCError_TO_STRING(ErrorID),
	OffMEssage := 	'OK',
	OffLevel := 	ADSLOG_MSGTYPE_HINT);

CalibrationEvent(
	Trigger :=	Calibrated,
	Level :=	ADSLOG_MSGTYPE_HINT,
	OnMessage := 'Focus is calibrated.'
	);

END_PROGRAM

// ---- POUs/FunctionBlocks/FB_Axis2.TcPOU
FUNCTION_BLOCK FB_Axis2
VAR_INPUT
	// enable the axis
	Enable:		BOOL;
	// reset the axis after error
	Reset: 		BOOL;
	// Move the Axis to a given position
	MoveAxis: 	BOOL;
	// HomeAxis;
	HomeAxis:	BOOL;
	// Stop the axis
	StopAxis:	BOOL;
	// position to move to
	Position: 	LREAL;
	// maximum velocity
	Velocity:	LREAL := 10.0;
	// Enable movement in positive direction (considering limit switch)
	Enable_Positive:	BOOL := TRUE;
	// Enable movement in negative direction (considering limit switch)
	Enable_Negative:	BOOL := TRUE;
	// jog forward
	Jog_Forward:		BOOL := FALSE;
	// jog backward
	Jog_Backwards:		BOOL := FALSE;
	// calibration input for homing
	bCalibrationCam:	BOOL;
	isModuloAxis:		BOOL := FALSE;
	// enable external setpoint generator
	Tracking:			BOOL;
	HomingMode:			MC_HomingMode := MC_HomingMode.MC_DefaultHoming;
END_VAR
VAR_OUTPUT
	// Reset has been executed
	ResetDone:	BOOL; 
	// the axis is in target position
	MoveDone:	BOOL;
	// the axis hass jogged
	JogDone:	BOOL;
	// the axis has stopped
	StopDone: 	BOOL;
	// the axis was calibrated and has come to a standstill
	HomeDone:	BOOL;
	// the axis is ready
	Ready:		BOOL;
	// the command has been aborted
	CommandAborted: BOOL;
	// axis busy
	Busy: 		BOOL;
	// axis is moving
	Active: 	BOOL;
	// axis is stopping
	Stopping:	BOOL;
	// axis is standing still (no commands issued) this should be the default
	StandStill:	BOOL;
	// axis is in motion
	InMotion:	BOOL;
	// axis is homing
	Homing:		BOOL;
	// axis is Accelerating or Decelerating
	InRamp:		BOOL;
	// axis is tracking on position
	isTracking:	BOOL;
	//	error condition
	Error: 		BOOL;
	// number of error
	ErrorID: 	UDINT;
	// actual position of the axis
	ActualPosition: LREAL;
	// axis is calibrated;
	Calibrated:	BOOL := FALSE;
	
END_VAR
VAR
	Axis_Power:		MC_Power;
	Axis_Reset:		MC_Reset;
	Axis_Move:		MC_MoveAbsolute;
	Axis_Modulo:	MC_MoveModulo;
	//Axis_Position:	MC_ReadActualPosition;
	Axis_Stop:		MC_Stop;
	Axis_Status:	MC_ReadStatus;
	Axis_Home:		MC_Home;
	Axis_Jog: 		MC_Jog;
	Axis_SetpointEnable:	MC_ExtSetPointGenEnable;
	Axis_SetpointDisable:	MC_ExtSetPointGenDisable;
	StopAllowed:	BOOL;
	// Direction for Axis_SetpointFeed
	Direction:			DINT;
	// difference between set position and measured position
	PositionDifference:	LREAL;
	TrackPosition:		LREAL;
	TrackVelocity:		LREAL;
	TrackAcceleration:	LREAL;
END_VAR

VAR_IN_OUT
	// axis reference
	AxisRef:	AXIS_REF;
END_VAR

// query the status of the axis at the beginning of the cycle
Axis_Status(Enable := TRUE,
			Axis := AxisRef);

// Enable the axis (power signal or manual enable)
Axis_Power(
	Axis := AxisRef,
	Enable := Enable,
	Enable_Positive := Enable_Positive,
	Enable_Negative := Enable_Negative,
	Override := 100.0,
	Status => Ready);

Axis_Reset(
	Axis := 	AxisRef,
	Execute := 	Reset,
	Done => 	ResetDone);

(* Tracking section ********************************************** *)

IF Tracking THEN
	PositionDifference := LIMIT(-0.002, Position - ActualPosition, 0.002);
	TrackPosition := ActualPosition + PositionDifference;
	TrackVelocity := 0.0; // LIMIT(-1.0, 2.0 * Velocity, 1.0);
	TrackAcceleration := 0.0;
ELSE
	TrackPosition := ActualPosition;
	TrackVelocity := 0.0;
	TrackAcceleration := 0.0;
END_IF


IF NOT Tracking OR ABS(PositionDifference) < 1E-5 THEN // TrackVelocity = 0 AND TrackAcceleration = 0 THEN
	Direction := 0;
ELSIF PositionDifference < 0.0 THEN
	Direction := -1;
ELSE
	Direction := 1;
END_IF

isTracking := Tracking AND ABS(Position - ActualPosition) < 5.0E-3;
IF Tracking AND Ready AND Calibrated AND NOT StopAxis THEN
	Axis_SetpointEnable.Execute := TRUE;
ELSIF NOT Axis_SetpointEnable.Busy AND Axis_SetpointEnable.Done THEN
	Axis_SetpointEnable.Execute := FALSE;
END_IF

Axis_SetpointEnable(Axis := AxisRef,
	Position :=		TrackPosition,	// final destination
	PositionType := POSITIONTYPE_ABSOLUTE);
	
MC_ExtSetPointGenFeed(
	Position :=		TrackPosition,
	Velocity :=		TrackVelocity,
	Acceleration :=	TrackAcceleration,
	Direction :=	Direction, 
	Axis :=			AxisRef);

Axis_SetpointDisable(Axis := AxisRef,
	Execute := NOT Tracking);
	
(* end of tracking section  ********************************************** *)
	
IF isModuloAxis THEN
	Axis_Modulo( 
		Axis := 		AxisRef,
		Execute := 		MoveAxis AND Ready AND Calibrated,
		Position := 	Position,
		Velocity :=		Velocity,
		Direction := 	MC_Shortest_Way,
		Done => 		MoveDone);
ELSE
	Axis_Move( 
		Axis := 		AxisRef,
		Execute := 		MoveAxis AND Ready AND Calibrated,
		Position := 	Position,
		Velocity := 	Velocity,
		Done => 		MoveDone);
END_IF

Axis_Jog(
	JogForward := 	Jog_Forward AND Ready AND Enable_Positive,
	JogBackwards := Jog_Backwards AND Ready AND Enable_Negative,
	Mode := 		MC_JOGMODE_STANDARD_FAST,
	Done => 		JogDone, 
	Axis := 		AxisRef);

Axis_Home(
	Axis := 			AxisRef,
	Execute := 			HomeAxis AND Ready,
	Position := 		position, //DEFAULT_HOME_POSITION,
	HomingMode :=		HomingMode,
	bCalibrationCam := 	bCalibrationCam,
	Done => 			HomeDone);	
(*	
IF (MoveDone OR HomeDone OR JogDone) AND NOT Axis_Status.StandStill THEN
	StopAxis := TRUE;
END_IF
*)
IF MoveDone AND (NOT Axis_Modulo.Busy OR NOT Axis_Move.Busy) THEN
	MoveAxis := FALSE;
END_IF

IF JogDone THEN
	Jog_Forward := FALSE;
	Jog_Backwards := FALSE;
END_IF

IF HomeDone THEN
	Calibrated := TRUE;
	HomeAxis := FALSE;
END_IF

IF StopDone THEN
	StopAxis := FALSE;
END_IF

StopAllowed :=	Axis_Status.StandStill OR  
				Axis_Status.ContinuousMotion OR
				Axis_Status.DiscreteMotion OR
				Axis_Status.SynchronizedMotion OR
				Axis_Status.Homing;

Axis_Stop( 
	Axis := 	AxisRef,
	Execute := 	StopAxis AND StopAllowed,
	Done => 	StopDone);
(*
Axis_Position(
	Axis := 	AxisRef,
	Enable := 	Calibrated,
	Position => AbsolutePosition);
*)
IF isModuloAxis THEN
	ActualPosition := AxisRef.NcToPlc.ModuloActPos; // required e.g. for Filterwheel
ELSE
	ActualPosition := AxisRef.NcToPlc.ActPos;
END_IF

IF Axis_Power.Error THEN
	ErrorID := Axis_Power.ErrorID;
END_IF

IF Axis_SetpointEnable.Error THEN
	ErrorID := Axis_SetpointEnable.ErrorID;
END_IF

IF Axis_Reset.Error THEN
	ErrorID := Axis_Reset.ErrorID;
END_IF

IF Axis_Modulo.Error THEN
	ErrorID := Axis_Modulo.ErrorID;
END_IF

IF Axis_Move.Error THEN
	ErrorID := Axis_Move.ErrorID;
END_IF

IF Axis_Home.Error THEN
	ErrorID := Axis_Home.ErrorID;
END_IF

IF Axis_Jog.Error THEN
	ErrorID := Axis_Jog.ErrorID;
END_IF

IF Axis_Stop.Error THEN
	ErrorID := Axis_Stop.ErrorID;
END_IF

Busy := 	Axis_SetpointEnable.Busy OR
			Axis_Reset.Busy OR 
			Axis_Modulo.Busy OR
			Axis_Move.Busy OR 
			Axis_Home.Busy OR
			Axis_Jog.Busy;

Error := 	Axis_Power.Error OR 
			Axis_SetpointEnable.Error OR
			Axis_Reset.Error OR 
			Axis_Modulo.Error OR
			Axis_Move.Error OR 
			Axis_Home.Error OR
			Axis_Jog.Error OR 
			Axis_Stop.Error;

Active := 	// Axis_Power.Active OR //alsways true if enabled 
			Axis_Modulo.Active OR
			Axis_Move.Active OR 
			Axis_Home.Active OR
			Axis_Jog.Active OR 
			Axis_Stop.Active;

CommandAborted :=	Axis_Modulo.CommandAborted OR
					Axis_Move.CommandAborted OR 
					Axis_Home.CommandAborted OR
					Axis_Jog.CommandAborted OR 
					Axis_Stop.CommandAborted;	
	
IF NOT Error THEN
	ErrorID := 0;
END_IF
			
InMotion := Axis_Status.ConstantVelocity OR
			Axis_Status.DiscreteMotion OR
			Axis_Status.ContinuousMotion OR
			Axis_Status.SynchronizedMotion; 
InRamp :=	Axis_Status.Accelerating OR
			Axis_Status.Decelerating;
Stopping := Axis_Status.Stopping;
StandStill := Axis_Status.StandStill;
Homing :=	Axis_Status.Homing;
// InPosition := AxisRef.NcToPlc.TargetPos;

END_FUNCTION_BLOCK

// ---- POUs/Functions/NCError_TO_STRING.TcPOU
FUNCTION NCError_TO_STRING : STRING(255)
VAR_INPUT
	// NC Error ID
	ErrorID:	UDINT;
END_VAR
VAR
END_VAR

NCError_TO_STRING := '';

CASE ErrorID OF
	16#4220:	NCError_TO_STRING := 'Group not ready / group not ready for new task';
	16#4253:	NCError_TO_STRING := 'Reference cam became free too soon';
	16#4260:	NCError_TO_STRING := 'Controller enable';
	16#42EF:	NCError_TO_STRING := 'Axis is locked for motion commands because a stop command is still active';
	16#4466:	NCError_TO_STRING := 'Invalid IO data FOR more than n subsequent NC cycles (encoder)';
	16#4550: 	NCError_TO_STRING := 'Following error monitoring (position)';
	16#4650:	NCError_TO_STRING := 'Drive hardware not ready to operate';
	16#4B07:	NCError_TO_STRING := 'Timeout axis function block';
	16#4B09:	NCError_TO_STRING := 'Axis is not ready';
	16#4B0A:	NCError_TO_STRING := 'Error during referencing';
	16#ECD0:	NCError_TO_STRING := 'Positive limit switch warning.';				
	16#ED43:	NCError_TO_STRING := 'Under-voltage - DC link.';				
	16#F601:	NCError_TO_STRING := 'Calibrate commutation offset error.';				

ELSE
	NCError_TO_STRING := DWORD_TO_HEXSTR(ErrorID, 4, FALSE);
END_CASE

END_FUNCTION

// ---- POUs/DerotatorControl.TcPOU
PROGRAM DerotatorControl
VAR_INPUT
	// enable the derotator
	enable:		BOOL;
	// reset an error
	reset:		BOOL;
	// decrease derotator angle
	left:		BOOL;
	// increase derotator angle
	right:		BOOL;
	// set the absolute position
	position:	LREAL;
	// derotator velocity
	Velocity:	LREAL := 10.0;
	// move to given position
	MoveAxis: 	BOOL;
	// calibrate the axis
	HomeAxis:	BOOL;
	// tracking flag
	Tracking:	BOOL;
	// stop the Axis
	StopAxis:	BOOL;
	// diagnostic error code reset
	bSoEReset: 			BOOL;
END_VAR
VAR_OUTPUT
	// error flag
	Error:				BOOL;
	// nc error id
	ErrorID:			UDINT;
	// actual position of the derotator
	actual_position:	LREAL;
	// calibrated flag
	Calibrated:			BOOL;
	// axis ready flag
	Ready:				BOOL;
	// position to move the axis to
	slewtime: 			LREAL;
END_VAR
VAR
	// trigger for the torque error
	TorqueError:		TON := (PT := T#3S);
	// axis function block
	DerotatorAxis:		FB_Axis2;
	
	DerotatorEvent:		FB_EventLog;
	// torque warning event
	TorqueWarning:		FB_EventLog;
	// torque calibration event
	CalibrationEvent:	FB_EventLog;
	// diagnostic low-level event
	DerotatorDiagnosticEvent: FB_EventLog;
	// percentage of the derotator torque
	derotator_torque:	REAL;
	// read slewtime
	ReadParameter:		MC_ReadParameter;
	fbSoEReset: 		FB_SoEReset;
	DiagnosticError:	BOOL;
END_VAR
VAR CONSTANT
	// current position of the calibration cam. Apply an offset here if necessary
	calibration_position:	LREAL := 438.4623; // calibration in positive direction (was 460.0)
END_VAR

(*
Selection 6
Homing in Endlage:

https://infosys.beckhoff.com/index.php?content=../content/1031/ax5000_usermanual/html/ax5000_homing_hardware_end_position.htm&id=12221
NC-Interface:
PlcToNc-Achsinterface, Bit 8 namens AcceptBlockedDriveSignal im nDeCtrlDWord

SPS-Interface:
TcNc-Lib, siehe SPS-Funktion AxisSetAcceptBlockedDriveSignal in der TwinCAT  PLC Library: NC.
*)

position := LIMIT(-70, position, 380);

IF enable AND NOT DerotatorAxis.Calibrated THEN
	HomeAxis := TRUE;
END_IF

IF DerotatorAxis.Calibrated THEN
	HomeAxis := FALSE;
	Calibrated := DerotatorAxis.Calibrated;
END_IF
	
IF HomeAxis THEN
	position := calibration_position;
END_IF

DeRotatorAxis(
	enable := 			enable,
	Reset := 			Reset,
	MoveAxis :=			MoveAxis,
	HomeAxis :=			HomeAxis,
	StopAxis :=			StopAxis,
	HomingMode :=		MC_ForceCalibration,
	Position := 		position, 
	Velocity :=			Velocity,
	Enable_Positive := 	NOT GVL_Telescope.Derotator_inputs.0,
	Enable_Negative := 	NOT GVL_Telescope.Derotator_inputs.1,
	Jog_Forward := 		right,
	Jog_Backwards := 	left,
	bCalibrationCam :=	GVL_Telescope.Derotator_inputs.0,
	isModuloAxis :=		FALSE,
	Tracking :=			Tracking,
	ActualPosition => 	actual_position,
	Error => 			Error,
	ErrorID => 			ErrorID,
	AxisRef :=			GVL_Telescope.DerotatorAxisRef);
	
IF DeRotatorAxis.MoveDone OR Reset OR Error THEN
	MoveAxis := FALSE;
END_IF

IF DeRotatorAxis.HomeDone OR Reset OR Error THEN
	HomeAxis := FALSE;
END_IF
	
IF DeRotatorAxis.ResetDone THEN
	reset := FALSE;
END_IF

IF DeRotatorAxis.StopDone THEN
	StopAxis := FALSE;
END_IF

DiagnosticError := FALSE;
IF GVL_Telescope.Derotator_diagnostic < 16#D012 AND GVL_Telescope.Derotator_diagnostic > 16#D014 THEN
	DiagnosticError := TRUE;
	ErrorID := GVL_Telescope.Derotator_diagnostic;
	bSoeReset := reset;
END_IF

Ready := DeRotatorAxis.Ready;

ReadParameter(	Axis := GVL_Telescope.DerotatorAxisRef, 
				Enable := DeRotatorAxis.InMotion, 
				ParameterNumber := MC_AxisParameter.AxisRemainingTimeToGo, 
				ReadMode := E_ReadMode.READMODE_CYCLIC);
				
IF ReadParameter.Valid THEN
	slewtime := ReadParameter.Value;
END_IF

IF bSoEReset THEN
	fbSoEReset(
		Axis := GVL_Telescope.DerotatorAxisRef,
		Execute := TRUE,
		Timeout := DEFAULT_ADS_TIMEOUT);
 	IF NOT fbSoEReset.Busy THEN
		fbSoEReset(Axis := GVL_Telescope.DerotatorAxisRef, Execute := FALSE);
		bSoEReset := FALSE;
		Reset := TRUE;
	END_IF
END_IF

derotator_torque := GVL_Telescope.Derotator_torque / 10.0;

TorqueError(IN := ABS(derotator_torque) > 12.0);

DerotatorEvent(	
	Trigger := 		Error, 
	Level := 		ADSLOG_MSGTYPE_ERROR,
	FormatString :=	'Derotator Axis Error: %s',
	OnMessage := 	NCError_TO_STRING(ErrorID),
	OffMEssage := 	'OK',
	OffLevel := 	ADSLOG_MSGTYPE_HINT);
	
DerotatorDiagnosticEvent(	
	Trigger := 		DiagnosticError, 
	Level := 		ADSLOG_MSGTYPE_ERROR,
	FormatString :=	'Derotator Axis Diagnostic Error: %s',
	OnMessage := 	NCError_TO_STRING(GVL_Telescope.Derotator_diagnostic));
	
TorqueWarning(	
	Trigger := 		TorqueError.Q, 
	Level := 		ADSLOG_MSGTYPE_WARN,
	FormatString :=	'%s',
	OnMessage := 	'Derotator torque is high.');

CalibrationEvent(	
	Trigger := 		Calibrated, 
	Level := 		ADSLOG_MSGTYPE_HINT,
	OnMessage := 	'Derotator is calibrated.');

END_PROGRAM

// ---- POUs/ElevationControl.TcPOU
PROGRAM ElevationControl
VAR_INPUT
	// enable the axis
	enable: 	BOOL;
	// reset an error
	reset:		BOOL;
	// increase the eleveation
	up:			BOOL;
	// decrease the elevation
	down:		BOOL;
	// set position of the axis in degrees
	position:	LREAL;
	// set the Velocity of the axis
	velocity:	LREAL;
	// move axis command
	MoveAxis:	BOOL;
	// calibrate the axis
	HomeAxis:	BOOL;
	// enable tracking
	Tracking:	BOOL;
	// stop the Axis
	StopAxis:	BOOL;
	// reset diagnostic errors
	bSoEReset:	 	BOOL;
END_VAR
VAR_OUTPUT
	// axis is ready to operate
	Ready:			BOOL;
	// drive error condition
	error: 			BOOL;
	// warning condition
	warning:		BOOL;
	// actual position of the elevation axis
	actual_position: 	LREAL;
	// error ID of the elevation axis
	ErrorID: 		UDINT;
	// axis is calibrated
	Calibrated:		BOOL;
	// time to reach target position
	slewtime:		LREAL;
END_VAR
VAR
	ElevationAxis:			FB_Axis2;
	ElevationCalibration: 	MC_SetPosition;
	fbSoEReset: 			FB_SoEReset;
	// delay until commutator angle is measured
	readydelay:				TON;
	// disable trigger for hydraulics
	enable_trigger:			F_TRIG;
	// store last position
	getlastposition:		BOOL := TRUE;
	ElevationAxisEvent: 	FB_Eventlog;
	ElevationDiagnosticEvent: 	FB_Eventlog;
	ElevationBrakeEvent: 	FB_Eventlog;
	HighElevationEvent: 	FB_Eventlog;
	LowElevationEvent:		FB_Eventlog;
	TorqueWarning:			FB_EventLog;
	CalibrationEvent:		FB_Eventlog;
	// elevation torque in percent
	elevation_torque: 		REAL;
	// timer to trigger a warning if torque is high
	torque_timer:			TON;
	ReadParameter:			MC_ReadParameter;
	DiagnosticError:		BOOL;
END_VAR
VAR CONSTANT
	// current position of the calibration cam. Apply an offset here if necessary
	calibration_position:	LREAL := 44.144; //44.139; //44.061; //43.806122; //42.1281; //43.000
END_VAR
VAR PERSISTENT
	last_position:	LREAL := -1.0;
END_VAR

// limit the position input to a sane value
position := LIMIT(0.0, position, 90.0);

//if we enable the axis, we have to open the brake first
IF Enable THEN
	IF NOT Calibrated THEN
		CoverControl.open := TRUE;
		IF CoverControl.isopen THEN
			HydraulicsControl.open_brake();
		END_IF
	ELSE
		HydraulicsControl.open_brake();
	END_IF
	
END_IF

enable_trigger(CLK := enable);
// close the brake on the falling edge of the enable signal
IF enable_trigger.Q THEN
	HydraulicsControl.close_brake();
END_IF

IF ElevationAxis.Calibrated OR Error THEN
	HomeAxis := FALSE;
END_IF

Calibrated := ElevationAxis.Calibrated;

IF HomeAxis THEN
	position := calibration_position;
	MoveAxis := FALSE;
	Tracking := FALSE;
END_IF

IF MoveAxis THEN
	Tracking := FALSE;
END_IF

// if NOT Enabled and ActVelo>1 then issue a warning
warning := NOT enable AND GVL_Telescope.ElevationAxisRef.NcToPlc.ActVelo>2.0;

// deactivate limit switches on homing
MC_SetAcceptBlockedDriveSignal(
	Axis := GVL_Telescope.ElevationAxisRef, 
	Enable := HomeAxis);
	
ElevationAxis(
	Enable := 			enable AND HydraulicsControl.brake_open,
	Reset := 			reset,
	MoveAxis :=			MoveAxis,
	HomeAxis :=			HomeAxis,
	StopAxis :=			StopAxis,
	Tracking :=			Tracking,
	Position := 		position, 
	Velocity :=			Velocity,
	Enable_Positive :=  GVL_Telescope.Elevation_inputs.0 OR HomeAxis,
	Enable_Negative := 	GVL_Telescope.Elevation_inputs.1,
	Jog_Forward :=		up,
	Jog_Backwards := 	down,
	bCalibrationCam :=	NOT GVL_Telescope.Elevation_inputs.0,
	ActualPosition => 	actual_position,
	Error => 			error,
	ErrorID => 			ErrorID,
	AxisRef :=			GVL_Telescope.ElevationAxisRef);

IF ElevationAxis.MoveDone THEN
	MoveAxis := FALSE;
END_IF

IF ElevationAxis.HomeDone THEN
	HomeAxis := FALSE;
END_IF
	
IF ElevationAxis.ResetDone THEN
	reset := FALSE;
END_IF

IF ElevationAxis.StopDone THEN
	StopAxis := FALSE;
END_IF

DiagnosticError := FALSE;
IF GVL_Telescope.Elevation_diagnostic < 16#D012 AND GVL_Telescope.Elevation_diagnostic > 16#D014 THEN
	DiagnosticError :=TRUE;
	ErrorID := GVL_Telescope.Elevation_diagnostic;
END_IF

ElevationCalibration(Axis := GVL_Telescope.ElevationAxisRef,
	Execute := getlastposition AND last_position>=0.0 AND NOT Calibrated,
	Position := last_position);

IF ElevationCalibration.Done THEN
	getlastposition := FALSE;
END_IF

IF Calibrated THEN
	last_position := actual_position;
END_IF

IF bSoEReset THEN
	last_position := -1.0;
	fbSoEReset(
		Axis := GVL_Telescope.ElevationAxisRef,
		Execute := TRUE,
		Timeout := DEFAULT_ADS_TIMEOUT);
 	IF NOT fbSoEReset.Busy THEN
		fbSoEReset(Axis := GVL_Telescope.ElevationAxisRef, Execute := FALSE);
		bSoEReset := FALSE;
		Reset := TRUE;
	END_IF
END_IF 

readydelay(IN :=  HydraulicsControl.brake_open, PT := T#6000MS, Q=> ready);

ReadParameter(	Axis := GVL_Telescope.ElevationAxisRef, 
				Enable := ElevationAxis.InMotion, 
				ParameterNumber := MC_AxisParameter.AxisRemainingTimeToGo, 
				ReadMode := E_ReadMode.READMODE_CYCLIC);
				
IF ReadParameter.Valid THEN
	slewtime := ReadParameter.Value;
END_IF

elevation_torque := GVL_Telescope.Elevation_torque / 10.0;
torque_timer(IN := ABS(elevation_torque) > 50.0, PT := T#1000MS);
		
ElevationAxisEvent(	Trigger := Error, 
				Level := ADSLOG_MSGTYPE_ERROR,
				FormatString := 'Elevation Axis Error: %s',
				OnMessage := NCError_TO_STRING(ErrorID));

ElevationDiagnosticEvent(	
	Trigger := 		DiagnosticError, 
	Level := 		ADSLOG_MSGTYPE_ERROR,
	FormatString :=	'Elevation Axis Diagnostic Error: %s',
	OnMessage := 	NCError_TO_STRING(GVL_Telescope.Elevation_diagnostic));

				
HighElevationEvent(	Trigger := Calibrated AND actual_position > 85.0, 
				Level := ADSLOG_MSGTYPE_WARN,
				FormatString := 'High Elevation: %s',
				OnMessage := LREAL_TO_FMTSTR(actual_position, 2, TRUE));

LowElevationEvent(	Trigger := Calibrated AND actual_position < 5.0, 
				Level := ADSLOG_MSGTYPE_WARN,
				FormatString := 'Low Elevation: %s',
				OnMessage := LREAL_TO_FMTSTR(actual_position, 2, TRUE));
				
ElevationBrakeEvent( Trigger := NOT enable AND HydraulicsControl.brake_open, 
				Level := ADSLOG_MSGTYPE_WARN,
				FormatString := '%s',
				OnMessage := 'Brake was opened without elevation axis enabled!'); 

TorqueWarning(	
	Trigger := torque_timer.Q, 
	Level := 		ADSLOG_MSGTYPE_WARN,
	FormatString :=	'%s',
	OnMessage := 	'Elevation torque is high.');
	
CalibrationEvent(
	Trigger :=	Calibrated,
	Level :=	ADSLOG_MSGTYPE_HINT,
	OnMessage := 'Elevation is calibrated.'
	);

END_PROGRAM

